(* CODESYS project SPT_Diagnostic.library
   Company: Beckhoff Automation LLC
   DefaultNamespace: SPT_Diagnostic
   Version: 3.3.8
   Placeholder: SPT Diagnostic
   Author: SPT
   Title: SPT Diagnostic

Project tree, tasks and I/O mapping:
  libraries: SPT Base Types, * (Beckhoff Automation LLC); SPT Event Logger, * (Beckhoff Automation LLC); Tc2_EtherCAT, * (Beckhoff Automation GmbH); Tc2_IoFunctions, * (Beckhoff Automation GmbH); Tc2_Standard, * (Beckhoff Automation GmbH); Tc2_System, * (Beckhoff Automation GmbH); Tc2_Utilities, * (Beckhoff Automation GmbH); Tc3_EventLogger, * (Beckhoff Automation GmbH); Tc3_Module, * (Beckhoff Automation GmbH)
  Device Diagnostic/
    DUT/
      data type ST_DeviceInfo
    function block FB_Component_Devices [ST]: Reset, CyclicLogic, CyclicLogic_EtherCat, Update, Initialize, DeviceInfo, LocalAmsNetId
  EtherCat Diagnostic/
    DUT/
      data type ST_EtherCatMaster_Command
      data type ST_EtherCatMaster_Config
      data type ST_EtherCatMaster_HMI
      data type ST_EtherCatMaster_Status
      data type ST_SyncUnitInfo
    function F_EtherCAT_VendorIDtoString [ST]
    function block FB_EtherCatMaster [ST]: CreateEvents, Monitoring, Reset, CyclicLogic, Update, GetSlaveNameByAddr, GetSyncUnitSlaveNames, LookupMasterDevState, LookupSlaveDevState, RaiseAlarmWithStringsAndFlags, RaiseWarningWithStringParameters, SlaveIsPartOfSyncUnit, FB_init, HMICommunication, Initialize, MasterState, SlaveState, EtherCatMasterInfo
    function block FB_EtherCatSyncUnits [ST]: CyclicLogic, SyncUnits, Update, LocalAmsNetId
  Interface/
    interface I_Diagnostic: Update
    interface I_EtherCatSyncUnits: SyncUnits
    interface I_SafetyBase: DependenceFB, OK, SafetyReset
    interface I_SafetyReset: Execute, PulseDuration
    interface I_SafetySimulation: SimulateSafetyDiag, SimulateSafetyState
  Project Information/
    function F_GetCompany [ST]
    function F_GetTitle [ST]
    function F_GetVersion [ST]
  Safety/
    Safety FBs Diagnostic/
      DUT/
        data type E_ComponentSafetyConnection_State
        data type E_ComponentSafetyEdm_State
        data type E_ComponentSafetyEStop_State
        data type E_ComponentSafetyGroup_Diag
        data type E_ComponentSafetyGroup_State
        data type E_ComponentSafetyMon_State
        data type E_ComponentSafetyOrAnd_State
        data type ST_SafetyStateDiag
      Reset Functionblocks/
        function block FB_SafetyResetPulse [ST]: CyclicLogic, Execute, PulseDuration
      function block FB_Component_Safety_AndOrFB [ST]: CyclicLogic, Initialize
      function block FB_Component_Safety_Base [ST]: Reset, CyclicLogic, DependenceFB, OK, SafetyReset, SimulateSafetyDiag, SimulateSafetyState, Initialize
      function block FB_Component_Safety_ConnectionFB [ST]: CreateEvents, Monitoring, Reset, CyclicLogic, Initialize
      function block FB_Component_Safety_EdmFB [ST]: CreateEvents, Monitoring, Reset, CyclicLogic, Initialize
      function block FB_Component_Safety_EstopFB [ST]: CreateEvents, Monitoring, Reset, CyclicLogic, ActiveName, Initialize
      function block FB_Component_Safety_Group [ST]: CreateEvents, Monitoring, Reset, CyclicLogic, AutoResetConnectionFaults, Initialize
      function block FB_Component_Safety_MonFB [ST]: CreateEvents, Monitoring, Reset, CyclicLogic, ActiveAlarm, ActiveName
    Safety Hardware Diagnostic/
  Version/
    global variables Global_Version
  global variables Parameter_Diagnostic
*)

// Device Diagnostic/DUT/ST_DeviceInfo
TYPE ST_DeviceInfo :
	STRUCT
		AmsNetID	   : T_AMSNETID;
		DeviceID	   : UINT;
		DeviceName	   : T_MAXSTRING;
		DeviceType	   : IODEVICETYPES;
		ipDiagnosticFB : I_Diagnostic;
	END_STRUCT
END_TYPE

// EtherCat Diagnostic/DUT/ST_EtherCatMaster_Command
TYPE ST_EtherCatMaster_Command :
	STRUCT
	END_STRUCT
END_TYPE

// EtherCat Diagnostic/DUT/ST_EtherCatMaster_Config
TYPE ST_EtherCatMaster_Config :
	STRUCT
		DeviceInfo : ST_DeviceInfo;
	END_STRUCT
END_TYPE

// EtherCat Diagnostic/DUT/ST_EtherCatMaster_HMI
TYPE ST_EtherCatMaster_HMI :
	STRUCT
		Config	: ST_EtherCatMaster_Config;
		Command : ST_EtherCatMaster_Command;
		Status	: ST_EtherCatMaster_Status;
	END_STRUCT
END_TYPE

// EtherCat Diagnostic/DUT/ST_EtherCatMaster_Status
TYPE ST_EtherCatMaster_Status :
	STRUCT
		EcSlavesState		: ARRAY[0..Parameter_Diagnostic.ETHERCAT_MASTER_SLAVE_MAX] OF ST_EcSlaveState;
		ConfiguredSlaveInfo : ARRAY[0..Parameter_Diagnostic.ETHERCAT_MASTER_SLAVE_MAX] OF ST_EcSlaveConfigData;
		EcSlaveTopologyInfo : ARRAY[0..Parameter_Diagnostic.ETHERCAT_MASTER_SLAVE_MAX] OF ST_TopologyDataEx;
	END_STRUCT
END_TYPE

// EtherCat Diagnostic/DUT/ST_SyncUnitInfo
TYPE ST_SyncUnitInfo :
	STRUCT
		Parent		   : T_MAXSTRING;
		Name		   : STRING(63);
		NumberOfSlaves : UINT;
		Slaves		   : ARRAY[1..Parameter_Diagnostic.ETHERCAT_MASTER_SYNC_UNIT_SLAVE_MAX] OF UINT;
	END_STRUCT
END_TYPE

// Safety/Safety FBs Diagnostic/DUT/E_ComponentSafetyConnection_State
{attribute 'qualified_only'}
{attribute 'strict'}
TYPE E_ComponentSafetyConnection_State : (
		Reset	   := 100,
		Session	   := 101,
		Connection := 102,
		Parameter  := 103,
		Data	   := 104,
		Shutdown   := 105,
		Deactive   := 106
	) USINT;
END_TYPE

// Safety/Safety FBs Diagnostic/DUT/E_ComponentSafetyEdm_State
{attribute 'qualified_only'}
TYPE E_ComponentSafetyEdm_State : (
		Invalid := 0,
		Stop	:= 2,
		Error	:= 4,
		Reset	:= 5,
		MonOff	:= 14,
		MonOn	:= 15
	) USINT;
END_TYPE

// Safety/Safety FBs Diagnostic/DUT/E_ComponentSafetyEStop_State
{attribute 'qualified_only'}
TYPE E_ComponentSafetyEStop_State : (
		Invalid	 := 0,
		Run		 := 1,
		Stop	 := 2,
		Safe	 := 3,
		Error	 := 4,
		Reset	 := 5,
		Start	 := 6,
		DelayOut := 7
	) USINT;
END_TYPE

// Safety/Safety FBs Diagnostic/DUT/E_ComponentSafetyGroup_Diag
{attribute 'qualified_only'}
TYPE E_ComponentSafetyGroup_Diag : (
		NoError		  := 0,
		FbError		  := 1,
		ComError	  := 2,
		ModuleError	  := 3,
		CmpError	  := 4,
		DeactiveError := 5,
		RestartError  := 6
	) UINT;
END_TYPE

// Safety/Safety FBs Diagnostic/DUT/E_ComponentSafetyGroup_State
{attribute 'qualified_only'}
TYPE E_ComponentSafetyGroup_State : (
		Invalid		 := 0,
		Run			 := 1,
		Stop		 := 2,
		Error		 := 4,
		Reset		 := 5,
		Start		 := 6,
		StopError	 := 7,
		Deactive	 := 16,
		WaitComError := 17
	) USINT;
END_TYPE

// Safety/Safety FBs Diagnostic/DUT/E_ComponentSafetyMon_State
{attribute 'qualified_only'}
TYPE E_ComponentSafetyMon_State : (
		Invalid	   := 0,
		Run		   := 1,
		Stop	   := 2,
		Safe	   := 3,
		Error	   := 4,
		Reset	   := 5,
		Start	   := 6,
		ErrorDelay := 7,
		DelayOut   := 8,
		FuncTest   := 9
	) USINT;
END_TYPE

// Safety/Safety FBs Diagnostic/DUT/E_ComponentSafetyOrAnd_State
{attribute 'qualified_only'}
TYPE E_ComponentSafetyOrAnd_State : (
		Invalid := 0,
		Run		:= 1,
		Stop	:= 2,
		Safe	:= 3
	) USINT;
END_TYPE

// Safety/Safety FBs Diagnostic/DUT/ST_SafetyStateDiag
{attribute 'pack_mode' := '1'}
TYPE ST_SafetyStateDiag :
	STRUCT
		State : USINT;
		Diag  : UINT; // **NOT PRESENT ON AND/OR FBs ** For components with USINT as Diag connection, connect first 8 Bit of UINT Diag. Inherited FB is evaluating correct length.
	END_STRUCT
END_TYPE

// Version/Global_Version
{attribute 'TcGenerated'}
{attribute 'no-analysis'}
{attribute 'linkalways'}
// This function has been automatically generated from the project information.
VAR_GLOBAL CONSTANT
	{attribute 'const_non_replaced'}
	stLibVersion_SPT_Diagnostic : ST_LibVersion := (iMajor := 3, iMinor := 3, iBuild := 8, iRevision := 0, nFlags := 1, sVersion := '3.3.8');
END_VAR

// Parameter_Diagnostic
{attribute 'qualified_only'}
VAR_GLOBAL CONSTANT
	UPDATE_TIME : TIME	:= T#500MS; // Start Diagnostic Run every xxx ms, T#0s = deactivated, update needs to manually occur via I_Diagnostic.Upadate()
	DEVICES_MAX : UDINT := 5;		// Max Devices in this System

	// EtherCat
	ETHERCAT_MASTER_START_UP_TIME		: TIME					  := T#1S; // Time to Startup EtherCat Master Diagnostic at initial startup
	ETHERCAT_MASTER_MAX					: UDINT					  := 5;	   // Max EtherCat Masters
	ETHERCAT_MASTER_SLAVE_MAX			: UDINT(1..EC_MAX_SLAVES) := 50;   // Max Slaves per EtherCat Master
	ETHERCAT_MASTER_SYNC_UNIT_MAX		: UDINT					  := 10;   // Max Count of Sync Units per Master
	ETHERCAT_MASTER_SYNC_UNIT_SLAVE_MAX : UDINT					  := 30;   // Max Count of Slaves per Sync Unit

	// Profinet

	// ProfiBus

	// EtherNet

	//...
END_VAR

// Device Diagnostic/FB_Component_Devices
{attribute 'no_explicit_call' := 'do not call this FB directly'}
FUNCTION_BLOCK FB_Component_Devices EXTENDS FB_ComponentBase IMPLEMENTS I_Diagnostic
VAR
	// System Information
	GetLocalAmsNetId : FB_GetLocalAmsNetId;
	GetDeviceIds	 : IOF_GetDeviceIDs;
	DeviceIds		 : ARRAY[0..Parameter_Diagnostic.DEVICES_MAX] OF WORD; //0 = Device counter, 1..X = Device ID's
	GetDeviceType	 : IOF_GetDeviceType;
	GetDeviceName	 : IOF_GetDeviceName;
	GetDeviceNetId	 : IOF_GetDeviceNetId;

	// Instances of Devices
	EtherCatSyncUnits	: FB_EtherCatSyncUnits;																		  // All Sync Units in this runtime
	EtherCatMaster		: ARRAY[1..Parameter_Diagnostic.ETHERCAT_MASTER_MAX] OF FB_EtherCatMaster(EtherCatSyncUnits); //
	EtherCatMasterCount : UDINT(0..Parameter_Diagnostic.ETHERCAT_MASTER_MAX) := 0;									  // Start at 0 to identify existing during Initialzation

	// Properties
	_DeviceInfo	   : ARRAY[1..Parameter_Diagnostic.DEVICES_MAX] OF ST_DeviceInfo;
	_LocalAmsNetId : T_AmsNetId := '';

	// Alarms

	// HMI

	// Sequences
	InitializeSequence : UDINT := 0;
	DeviceNumber	   : UDINT := 1;
	i				   : UDINT := 0; // Iterator
END_VAR

VAR
	// Local
	UpdateOn	: TON;
	UpdateOff	: TON;
	RtrigUpdate : R_TRIG;
END_VAR

//! @summary Clears error flags and error IDs for this component
METHOD PUBLIC Reset : BOOL
Reset := SUPER^.Reset();
IF EtherCatMasterCount >= 1 THEN
	FOR i := 1 TO EtherCatMasterCount DO
		EtherCatMaster[i].Reset();
	END_FOR
END_IF
END_METHOD

//! @summary This method serves as the entry point for all underlying FB logic
METHOD PUBLIC CyclicLogic

//! @description This method should be called cyclically by descendant function blocks by invoking <c>SUPER^.CyclicLogic()</c>.  Alternatively, the contents of this method could be reimplemented entirely in which case a call to this method would not be necessary.
IF NOT _InitComplete THEN
	_InitComplete := Initialize();
	RETURN;
END_IF

// Update Toggle
IF Parameter_Diagnostic.UPDATE_TIME > T#0MS THEN
	UpdateOn(IN := NOT UpdateOff.Q, PT := Parameter_Diagnostic.UPDATE_TIME);
	UpdateOff(IN := UpdateOn.Q, PT := Parameter_Diagnostic.UPDATE_TIME);
	RtrigUpdate(CLK := UpdateOn.Q);
END_IF

// Cyclic Logics
CyclicLogic_EtherCat();
SUPER^.CyclicLogic();

// Error Status Update of all Devices
_Error := FALSE;
_Busy  := FALSE;
IF EtherCatMasterCount >= 1 THEN
	FOR i := 1 TO EtherCatMasterCount DO
		IF _CurrentAlarmSeverity < EtherCatMaster[i].CurrentAlarmSeverity THEN
			_CurrentAlarmSeverity := EtherCatMaster[i].CurrentAlarmSeverity;
		END_IF

		_Error := _Error OR EtherCatMaster[i].Error;
		_Busy  := _Busy OR EtherCatMaster[i].Busy;
		IF EtherCatMaster[i].ErrorID <> 0 AND _ErrorID = 0 THEN
			_ErrorID := EtherCatMaster[i].ErrorID;
		END_IF
	END_FOR
END_IF
END_METHOD

METHOD CyclicLogic_EtherCat
// Get all Sync Units in Runtime
EtherCatSyncUnits.LocalAmsNetId := _LocalAmsNetId;
EtherCatSyncUnits.CyclicLogic();

// Call Cyclic
IF EtherCatMasterCount >= 1 THEN
	FOR i := 1 TO EtherCatMasterCount DO
		// Update
		IF RtrigUpdate.Q THEN
			EtherCatMaster[i].Update();
		END_IF

		// Cyclic Call
		EtherCatMaster[i].CyclicLogic();
	END_FOR
END_IF
END_METHOD

METHOD Update
IF EtherCatMasterCount >= 1 THEN
	FOR i := 1 TO EtherCatMasterCount DO
		EtherCatMaster[i].Update();
	END_FOR
END_IF
END_METHOD

//! @summary Basic component initialization logic
METHOD PROTECTED Initialize : BOOL;
//! @description This method is called by <c>CyclicLogic()</c> as required
VAR_INST
	AllDevicesInitialized : BOOL := FALSE;
END_VAR
Initialize := FALSE;
IF _Simulate THEN
	Initialize := SUPER^.Initialize();
	RETURN;
END_IF

// Call FBs
GetLocalAmsNetId(tTimeOut := T#1S);
GetDeviceIds(NETID := _LocalAmsNetId, TMOUT := T#1S);
GetDeviceName(NETID := _LocalAmsNetId, TMOUT := T#1S);
GetDeviceNetId(NETID := _LocalAmsNetId, TMOUT := T#1S);
GetDeviceType(NETID := _LocalAmsNetId, TMOUT := T#1S);

// Init Sequence
CASE InitializeSequence OF
	0: // Get local AmsNet-Id
		GetLocalAmsNetId.bExecute := TRUE;
		IF GetLocalAmsNetId.bBusy THEN
			InitializeSequence := InitializeSequence + 10;
		END_IF

	10: // Get local AmsNet-Id
		IF NOT GetLocalAmsNetId.bBusy AND NOT GetLocalAmsNetId.bError THEN
			_LocalAmsNetId	   := GetLocalAmsNetId.AddrString;
			InitializeSequence := InitializeSequence + 10;
		END_IF

		IF GetLocalAmsNetId.bError THEN
			_ErrorID := GetLocalAmsNetId.nErrId;
			Trace('Init Failed - GetLocalAmsNetId!');
			InitializeSequence := 999;
		END_IF

	20: // Get all Devices in this System
		GetDeviceIds.LEN	  := SIZEOF(DeviceIds);
		GetDeviceIds.DESTADDR := ADR(DeviceIds);
		GetDeviceIds.START	  := TRUE;
		IF GetDeviceIds.BUSY THEN
			GetDeviceIds.START := FALSE;
			InitializeSequence := InitializeSequence + 10;
		END_IF

	30: // Get all Devices in this System
		IF NOT GetDeviceIds.BUSY AND NOT GetDeviceIds.ERR THEN
			// Devices found
			IF (DeviceIDs[0] > 0) AND NOT _Simulate THEN
				// Map device Ids
				FOR i := 1 TO DeviceIDs[0] DO
					IF i <= Parameter_Diagnostic.DEVICES_MAX THEN
						_DeviceInfo[i].DeviceID := DeviceIDs[i];
					ELSE
						Trace('Init Failed - find IO Devices, Diagnostic, not enough Devices foreseen! Increase DEVICES_MAX');
						InitializeSequence := 999;
						EXIT;
					END_IF
				END_FOR

				InitializeSequence := InitializeSequence + 10;
			ELSE
				_Simulate		   := TRUE; // No devices found = activate simulation mode
				InitializeSequence := 1000;
			END_IF
		END_IF

		IF GetDeviceIds.ERR THEN
			_ErrorID := GetDeviceIds.ERRID;
			Trace('Init Failed - GetDeviceIds!');
			InitializeSequence := 999;
		END_IF

	40: // Get Device Names
		GetDeviceName.DEVICEID := DeviceIDs[DeviceNumber];
		GetDeviceName.START	   := TRUE;
		IF GetDeviceName.BUSY THEN
			GetDeviceName.START := FALSE;
			InitializeSequence	:= InitializeSequence + 10;
		END_IF

	50: // Get Device Names
		IF NOT GetDeviceName.BUSY AND NOT GetDeviceName.ERR THEN
			// Next Device
			_DeviceInfo[DeviceNumber].DeviceName := GetDeviceName.DEVICENAME;
			DeviceNumber						 := DeviceNumber + 1;
			IF (DeviceIDs[DeviceNumber] <> 0) THEN
				InitializeSequence := InitializeSequence - 10;
			ELSE
				DeviceNumber	   := 1;
				InitializeSequence := InitializeSequence + 10;
			END_IF
		END_IF

		IF GetDeviceName.ERR THEN
			_ErrorID := GetDeviceName.ERRID;
			Trace('Init Failed - GetDeviceName!');
			InitializeSequence := 999;
		END_IF

	60: // Get Device NetIds
		GetDeviceNetId.DEVICEID := DeviceIDs[DeviceNumber];
		GetDeviceNetId.START	:= TRUE;
		IF GetDeviceNetId.BUSY THEN
			GetDeviceNetId.START := FALSE;
			InitializeSequence	 := InitializeSequence + 10;
		END_IF

	70: // Get Device NetIds
		IF NOT GetDeviceNetId.BUSY AND NOT GetDeviceNetId.ERR THEN
			// Next Device
			_DeviceInfo[DeviceNumber].AmsNetID := GetDeviceNetId.DeviceNetId;
			DeviceNumber					   := DeviceNumber + 1;
			IF (DeviceIDs[DeviceNumber] <> 0) THEN
				InitializeSequence := InitializeSequence - 10;
			ELSE
				DeviceNumber	   := 1;
				InitializeSequence := InitializeSequence + 10;
			END_IF
		END_IF

		IF GetDeviceNetId.ERR THEN
			_ErrorID := GetDeviceNetId.ERRID;
			Trace('Init Failed - GetDeviceNetId!');
			InitializeSequence := 999;
		END_IF

	80: // Get Device Types
		GetDeviceType.DEVICEID := DeviceIDs[DeviceNumber];
		GetDeviceType.START	   := TRUE;
		IF GetDeviceType.BUSY THEN
			GetDeviceType.START := FALSE;
			InitializeSequence	:= InitializeSequence + 10;
		END_IF

	90: // Get Device Types
		IF NOT GetDeviceType.BUSY AND NOT GetDeviceType.ERR THEN
			// Next Device
			_DeviceInfo[DeviceNumber].DeviceType := GetDeviceType.IODeviceType;
			DeviceNumber						 := DeviceNumber + 1;
			IF (DeviceIDs[DeviceNumber] <> 0) THEN
				InitializeSequence := InitializeSequence - 10;
			ELSE
				DeviceNumber	   := 1;
				InitializeSequence := InitializeSequence + 10;
			END_IF
		END_IF

		IF GetDeviceType.ERR THEN
			_ErrorID := GetDeviceType.ERRID;
			Trace('Init Failed - GetDeviceType!');
			InitializeSequence := 999;
		END_IF

	100: // Initalize all Devices found
		FOR i := 1 TO DeviceIDs[0] DO
			CASE DeviceInfo[i].DeviceType OF
				IODEVICETYPES.IODEVICETYPE_ETHERCAT:
					EtherCatMasterCount := EtherCatMasterCount + 1;
					IF EtherCatMasterCount <= Parameter_Diagnostic.ETHERCAT_MASTER_MAX THEN
						EtherCatMaster[EtherCatMasterCount].EtherCatMasterInfo REF= _DeviceInfo[i];
						EtherCatMaster[EtherCatMasterCount].Name			   := DeviceInfo[i].DeviceName;
						DeviceInfo[i].ipDiagnosticFB						   := EtherCatMaster[EtherCatMasterCount];
					ELSE
						Trace('Init Failed - not enough EtherCat Master Diagnostics Instances! Increase ETHERCAT_MASTER_MAX');
						InitializeSequence := 999;
					END_IF

			ELSE
				Trace(CONCAT('Warning - Device Diagnostics for this Device does not exist! ', DeviceInfo[i].DeviceName));
			END_CASE
		END_FOR

		// No error during initialization
		IF InitializeSequence <> 999 THEN
			InitializeSequence := InitializeSequence + 10;
		END_IF

	110: // Initalize all Devices found
		AllDevicesInitialized := TRUE;

		// Init all EtherCat Master Devices
		IF EtherCatMasterCount >= 1 THEN
			FOR i := 1 TO EtherCatMasterCount DO
				EtherCatMaster[i].CyclicLogic();
				AllDevicesInitialized := AllDevicesInitialized AND EtherCatMaster[i].InitComplete;
			END_FOR
		END_IF

		IF AllDevicesInitialized THEN
			InitializeSequence := 1000;
		END_IF

	1000: // Initialize the Base
		IF SUPER^.Initialize() THEN
			Initialize := TRUE;
			_Error	   := FALSE;
			_Busy	   := FALSE;
		END_IF

	999:
		_Error := TRUE;
		_Busy  := FALSE;
END_CASE
END_METHOD

{analysis -29}
PROPERTY DeviceInfo : REFERENCE TO ARRAY[1..Parameter_Diagnostic.DEVICES_MAX] OF ST_DeviceInfo
GET
DeviceInfo REF= _DeviceInfo;
END_GET
END_PROPERTY

PROPERTY LocalAmsNetId : T_AmsNetId
GET
LocalAmsNetId := _LocalAmsNetId;
END_GET
END_PROPERTY

END_FUNCTION_BLOCK

// Interface/I_Diagnostic
INTERFACE I_Diagnostic EXTENDS I_BaseFB

METHOD Update
VAR_INPUT
END_VAR
END_METHOD

END_INTERFACE

// EtherCat Diagnostic/FB_EtherCatSyncUnits
{attribute 'no_explicit_call' := 'do not call this FB directly'}
FUNCTION_BLOCK FB_EtherCatSyncUnits EXTENDS FB_CyclicFB IMPLEMENTS I_EtherCatSyncUnits
VAR
	(* Sequence *)
	SyncUnitSequence : UINT;

	(* Local *)
	GetSyncUnitOids			  : ADSRDWRT;
	GetAllSyncUnitSlaveAddr	  : FB_EcGetAllSyncUnitSlaveAddr;
	ipSyncUnitComObject		  : ITComObject;
	ipSyncUnitParentComObject : ITComObject;
	SyncUnitCount			  : DWORD;
	i						  : DWORD; // Iterator
	SyncUnitParentOid		  : OTCID;
	SyncUnitOids			  : ARRAY[1..Parameter_Diagnostic.ETHERCAT_MASTER_SYNC_UNIT_MAX] OF OTCID;

	(* Properties *)
	_SyncUnits	   : ARRAY[1..Parameter_Diagnostic.ETHERCAT_MASTER_SYNC_UNIT_MAX] OF ST_SyncUnitInfo;
	_LocalAmsNetId : T_AmsNetId;
END_VAR

VAR CONSTANT
	SYNC_UNIT_CLASS_ID : CLSID := STRING_TO_GUID('03020004-0000-0000-F000-000000000064');
END_VAR

METHOD PUBLIC CyclicLogic
VAR_INST
	tempName		 : STRING(63);
	SyncUnitIterator : UINT := 1;
END_VAR
{analysis -19}
{analysis -07}

// Call FBs
GetSyncUnitOids(NETID := _LocalAmsNetId);
GetAllSyncUnitSlaveAddr(sNetId := _LocalAmsNetId);

// Sequence
CASE SyncUnitSequence OF
	0: // Wait for start
		GetSyncUnitOids.WRTRD			 := FALSE;
		GetAllSyncUnitSlaveAddr.bExecute := FALSE;
		SyncUnitIterator				 := 1;

	10: // Get Sync Unit Count

		// Reset for restart
		_Error	 := FALSE;
		_ErrorID := 0;

		// Get Sync Unit Count
		GetSyncUnitOids.PORT	 := 10;
		GetSyncUnitOids.IDXGRP	 := 16#201;
		GetSyncUnitOids.IDXOFFS	 := 16#01;
		GetSyncUnitOids.WRITELEN := SIZEOF(SYNC_UNIT_CLASS_ID);
		GetSyncUnitOids.SRCADDR	 := ADR(SYNC_UNIT_CLASS_ID);
		GetSyncUnitOids.READLEN	 := SIZEOF(SyncUnitCount);
		GetSyncUnitOids.DESTADDR := ADR(SyncUnitCount);
		GetSyncUnitOids.WRTRD	 := TRUE;
		IF GetSyncUnitOids.BUSY THEN
			SyncUnitSequence := SyncUnitSequence + 10;
		END_IF

	20: // Get Sync Unit Count
		IF NOT GetSyncUnitOids.BUSY AND NOT GetSyncUnitOids.ERR THEN
			// Byte Adjustment
			SyncUnitCount		  := SyncUnitCount / 4;
			GetSyncUnitOids.WRTRD := FALSE;
			IF SyncUnitCount <= Parameter_Diagnostic.ETHERCAT_MASTER_SYNC_UNIT_MAX THEN // Check configuration and space
				IF SyncUnitCount > 0 THEN												// Only if Sync Unit exist - run diag
					SyncUnitSequence := SyncUnitSequence + 10;
				ELSE
					SyncUnitSequence := 0;
				END_IF
			ELSE
				SyncUnitSequence := 999;
				_ErrorID		 := SyncUnitCount;
				Trace('FB_EtherCatSyncUnits - not enough Sync Units foreseen! Increase ETHERCAT_MASTER_SYNC_UNIT_MAX');
			END_IF
		END_IF

		IF GetSyncUnitOids.ERR THEN
			_ErrorID		 := GetSyncUnitOids.ERRID;
			SyncUnitSequence := 999;
		END_IF

	30: // Get Sync Unit Oids
		GetSyncUnitOids.PORT	 := 10;
		GetSyncUnitOids.IDXGRP	 := 16#201;
		GetSyncUnitOids.IDXOFFS	 := 16#02;
		GetSyncUnitOids.WRITELEN := SIZEOF(SYNC_UNIT_CLASS_ID);
		GetSyncUnitOids.SRCADDR	 := ADR(SYNC_UNIT_CLASS_ID);
		GetSyncUnitOids.READLEN	 := (SIZEOF(OTCID) * SyncUnitCount);
		GetSyncUnitOids.DESTADDR := ADR(SyncUnitOids);
		GetSyncUnitOids.WRTRD	 := TRUE;
		IF GetSyncUnitOids.BUSY THEN
			SyncUnitSequence := SyncUnitSequence + 10;
		END_IF

	40: // Get Sync Unit Oids
		IF NOT GetSyncUnitOids.BUSY AND NOT GetSyncUnitOids.ERR THEN
			GetSyncUnitOids.WRTRD := FALSE;
			SyncUnitSequence	  := SyncUnitSequence + 10;
		END_IF

		IF GetSyncUnitOids.ERR THEN
			_ErrorID		 := GetSyncUnitOids.ERRID;
			SyncUnitSequence := 999;
		END_IF

	50: // Get EtherCat Master and Name of Sync Unit
		FOR i := 1 TO SyncUnitCount DO
			// Get Sync Unit
			FW_ObjMgr_GetObjectInstance(SyncUnitOids[i], TC_GLOBAL_IID_LIST.IID_ITComObject, ADR(ipSyncUnitComObject));
			IF ipSyncUnitComObject <> 0 THEN
				ipSyncUnitComObject.TcGetObjectName(objName := ADR(_SyncUnits[i].Name), nameLen := SIZEOF(_SyncUnits[i].Name));
				F_EcGetSyncUnitName(SyncUnitOids[i], sSyncUnitName => tempName);
				tempName		   := CONCAT(tempName, ' - ');
				_SyncUnits[i].Name := CONCAT(tempName, _SyncUnits[i].Name);

				// Get Parent
				ipSyncUnitComObject.TcGetParentObjId(SyncUnitParentOid);
				FW_ObjMgr_GetObjectInstance(SyncUnitParentOid, TC_GLOBAL_IID_LIST.IID_ITComObject, ADR(ipSyncUnitParentComObject));
				IF ipSyncUnitParentComObject <> 0 THEN
					ipSyncUnitParentComObject.TcGetObjectName(objName := ADR(_SyncUnits[i].Parent), nameLen := SIZEOF(_SyncUnits[i].Parent));
					FW_SafeRelease(pipUnk := ADR(ipSyncUnitParentComObject));
				END_IF

				FW_SafeRelease(pipUnk := ADR(ipSyncUnitComObject));
			END_IF
		END_FOR

		SyncUnitSequence := SyncUnitSequence + 10;

	60: // Get all sync Unit Slaves 
		IF SyncUnitIterator > Parameter_Diagnostic.ETHERCAT_MASTER_SYNC_UNIT_MAX THEN
			SyncUnitSequence := 0; // All Sync units searched
		ELSE
			IF SyncUnitOids[SyncUnitIterator] = 0 THEN
				SyncUnitSequence := 0; // Done
			ELSE
				GetAllSyncUnitSlaveAddr.nObjectId := SyncUnitOids[SyncUnitIterator];
				GetAllSyncUnitSlaveAddr.pAddrBuf  := ADR(_SyncUnits[SyncUnitIterator].Slaves);
				GetAllSyncUnitSlaveAddr.cbBufLen  := SIZEOF(_SyncUnits[SyncUnitIterator].Slaves);
				GetAllSyncUnitSlaveAddr.bExecute  := TRUE;
				IF GetAllSyncUnitSlaveAddr.bBusy THEN
					GetAllSyncUnitSlaveAddr.bExecute := FALSE;
					SyncUnitSequence				 := SyncUnitSequence + 10;
				END_IF
			END_IF
		END_IF

	70: // Get all sync Unit Slaves
		IF NOT GetAllSyncUnitSlaveAddr.bBusy AND NOT GetAllSyncUnitSlaveAddr.bError THEN
			_SyncUnits[SyncUnitIterator].NumberOfSlaves := GetAllSyncUnitSlaveAddr.nSlaves;
			SyncUnitIterator							:= SyncUnitIterator + 1;
			IF _SyncUnits[SyncUnitIterator].NumberOfSlaves <= Parameter_Diagnostic.ETHERCAT_MASTER_SYNC_UNIT_SLAVE_MAX THEN
				SyncUnitSequence := SyncUnitSequence - 10;
			ELSE
				SyncUnitSequence := 999;
				_ErrorID		 := _SyncUnits[SyncUnitIterator].NumberOfSlaves;
				Trace('FB_EtherCatSyncUnits - not enough slaves per Sync Units foreseen! Increase ETHERCAT_MASTER_SYNC_UNIT_SLAVE_MAX');
			END_IF
		END_IF

		IF GetAllSyncUnitSlaveAddr.bError THEN
			_ErrorID		 := GetAllSyncUnitSlaveAddr.nErrId;
			SyncUnitSequence := 999;
		END_IF

	999: // Error
		SyncUnitSequence := 0;
		_Error			 := TRUE;
		Trace('FB_EtherCatSyncUnits - Error get Sync Units Sequence!');
END_CASE

_Busy := SyncUnitSequence <> 0;
END_METHOD

PROPERTY SyncUnits : REFERENCE TO ARRAY[1..Parameter_Diagnostic.ETHERCAT_MASTER_SYNC_UNIT_MAX] OF ST_SyncUnitInfo
GET
SyncUnits REF= _SyncUnits;
END_GET
END_PROPERTY

METHOD Update
IF NOT _Busy THEN
	SyncUnitSequence := 10;
END_IF
END_METHOD

PROPERTY LocalAmsNetId : T_AmsNetId
SET
_LocalAmsNetId := LocalAmsNetId;
END_SET
END_PROPERTY

END_FUNCTION_BLOCK

// Interface/I_EtherCatSyncUnits
INTERFACE I_EtherCatSyncUnits EXTENDS I_Diagnostic

PROPERTY SyncUnits : REFERENCE TO ARRAY[1..Parameter_Diagnostic.ETHERCAT_MASTER_SYNC_UNIT_MAX] OF ST_SyncUnitInfo
GET
END_GET
END_PROPERTY

END_INTERFACE

// EtherCat Diagnostic/FB_EtherCatMaster
{attribute 'no_explicit_call' := 'do not call this FB directly'}
FUNCTION_BLOCK FB_EtherCatMaster EXTENDS FB_ComponentBase IMPLEMENTS I_Diagnostic
VAR
	(* Internal Variables *)
	EcGetMasterDevState	 : FB_EcGetMasterDevState;
	GetSlaveTopologyInfo : FB_EcGetSlaveTopologyInfo;
	EcGetAllSlaveStates	 : FB_EcGetAllSlaveStates;
	GetConfiguredSlaves	 : FB_EcGetConfSlaves;
	EcSlavesState		 : ARRAY[0..Parameter_Diagnostic.ETHERCAT_MASTER_SLAVE_MAX] OF ST_EcSlaveState;
	ConfiguredSlaveInfo	 : ARRAY[0..Parameter_Diagnostic.ETHERCAT_MASTER_SLAVE_MAX] OF ST_EcSlaveConfigData;
	EcSlaveTopologyInfo	 : ARRAY[0..Parameter_Diagnostic.ETHERCAT_MASTER_SLAVE_MAX] OF ST_TopologyDataEx;
	SyncUnits			 : REFERENCE TO ARRAY[1..Parameter_Diagnostic.ETHERCAT_MASTER_SYNC_UNIT_MAX] OF ST_SyncUnitInfo;
	MasterDevState		 : WORD;
	SlaveCount			 : UINT;
	CfgSlaveCount		 : UINT;

	(* Properties *)
	_EtherCatMasterInfo : REFERENCE TO ST_DeviceInfo;

	(* HMI *)
	EtherCatMaster_HMI : ST_EtherCatMaster_HMI;

	(* Sync Units *)
	ipEtherCatSyncUnits : I_EtherCatSyncUnits;

	(* Sequence *)
	SlaveSeq	: UINT;
	MasterSeq	: UINT;
	SyncUnitSeq : UINT;

	(* Alarms *)
	MasterAlarms	 : ARRAY[1..MASTER_ALARM_COUNT] OF FB_TcAlarm;
	SlaveErrors		 : ARRAY[0..Parameter_Diagnostic.ETHERCAT_MASTER_SLAVE_MAX] OF FB_TcAlarm;
	SlaveWarnings	 : ARRAY[0..Parameter_Diagnostic.ETHERCAT_MASTER_SLAVE_MAX] OF FB_TcAlarm;
	SyncUnitWarnings : ARRAY[1..Parameter_Diagnostic.ETHERCAT_MASTER_SYNC_UNIT_MAX] OF FB_TcAlarm;
END_VAR

VAR CONSTANT
	MASTER_ALARM_COUNT : UDINT := 3;
	STRING_LEN		   : INT   := 80;
END_VAR

METHOD PROTECTED CreateEvents
//! @description This method is called by <c>Initialize()</c> as required
VAR_INST
	tempName   : STRING;
	SourceInfo : FB_TcSourceInfo;
	i		   : UDINT;
END_VAR
F_CreateAllEventsInClass(Alarms		:= MasterAlarms,
						 ClassSize	:= SIZEOF(TC_EVENTS.EtherCatMaster),
						 pInitEvent := ADR(TC_EVENTS.EtherCatMaster.InitReferenceEvent),
						 Prefix		:= Name);

SUPER^.CreateEvents();

// Create SyncUnit and Slave Alarms
FOR i := 0 TO Parameter_Diagnostic.ETHERCAT_MASTER_SLAVE_MAX DO
	SourceInfo.sName := CONCAT(CONCAT(THIS^.Name, ' - '), ConfiguredSlaveInfo[i].sName);
	SlaveErrors[i].CreateEx(stEventEntry := TC_EVENTS.EtherCatSlave.SlaveError, 0, SourceInfo);
	SlaveWarnings[i].CreateEx(stEventEntry := TC_EVENTS.EtherCatSlave.SlaveWarning, 0, SourceInfo);
END_FOR

FOR i := 1 TO Parameter_Diagnostic.ETHERCAT_MASTER_SYNC_UNIT_MAX DO
	SourceInfo.sName := CONCAT(CONCAT(THIS^.Name, ' - '), ConfiguredSlaveInfo[i].sName);
	SyncUnitWarnings[i].CreateEx(stEventEntry := TC_EVENTS.SyncUnit.SyncUnitWarning, 0, SourceInfo);
END_FOR
END_METHOD

//! Provides basic error detection and event handling for this component
METHOD PROTECTED Monitoring
(*! @descriptionThis method is called cyclically by <c>CyclicLogic()</c>*)
VAR_INST
	Error1 : BOOL;
	Error2 : BOOL;
	Error3 : BOOL;
END_VAR
SUPER^.Monitoring();

(* EtherCat Master Messages *)

// Raised in Master Sequence

(* EtherCat Slave Messages *)

// Raised in Slave Sequence

(* Alarm Severity of EtherCat Master Device *)
_CurrentAlarmSeverity := F_GetMaxSeverityRaised(Alarms := MasterAlarms, CurrentSeverity := _CurrentAlarmSeverity);
_CurrentAlarmSeverity := F_GetMaxSeverityRaised(Alarms := SlaveErrors, CurrentSeverity := _CurrentAlarmSeverity);
_CurrentAlarmSeverity := F_GetMaxSeverityRaised(Alarms := SlaveWarnings, CurrentSeverity := _CurrentAlarmSeverity);
_CurrentAlarmSeverity := F_GetMaxSeverityRaised(Alarms := SyncUnitWarnings, CurrentSeverity := _CurrentAlarmSeverity);
END_METHOD

//! @summary Clears error flags and error IDs for this component
METHOD PUBLIC Reset : BOOL
F_ClearAllEventsInClass(MasterAlarms);
F_ClearAllEventsInClass(SlaveErrors);
F_ClearAllEventsInClass(SlaveWarnings);
F_ClearAllEventsInClass(SyncUnitWarnings);
SlaveSeq  := 0;
MasterSeq := 0;
_Error	  := FALSE;
_ErrorID  := 0;
_Busy	  := FALSE;
Reset	  := SUPER^.Reset();
END_METHOD

//! @summary This method serves as the entry point for all underlying FB logic
METHOD PUBLIC CyclicLogic

//! @description This method should be called cyclically by descendant function blocks by invoking <c>SUPER^.CyclicLogic()</c>.  Alternatively, the contents of this method could be reimplemented entirely in which case a call to this method would not be necessary.
IF NOT _InitComplete THEN
	_InitComplete := Initialize();
	RETURN;
END_IF

(* Main Component Signals *)
IF _Simulate THEN
	_Busy	 := FALSE;
	_Error	 := FALSE;
	_ErrorID := 0;
ELSE
	// Master State
	MasterState();

	// Slave State
	SlaveState();

	// Super
	_Busy := SlaveSeq <> 0 OR MasterSeq <> 0; // Sequence running
	SUPER^.CyclicLogic();
END_IF
END_METHOD

METHOD Update
IF NOT _Busy THEN
	// Start Master and Slave Diagnostics Sequence
	MasterSeq := 10;
	SlaveSeq  := 10;
END_IF
END_METHOD

METHOD PRIVATE GetSlaveNameByAddr : STRING(31)
VAR_INPUT
	Addr : UINT;
END_VAR

VAR_INST
	Slave : UDINT;
END_VAR
GetSlaveNameByAddr := '';
FOR Slave := 0 TO Parameter_Diagnostic.ETHERCAT_MASTER_SLAVE_MAX DO
	IF ConfiguredSlaveInfo[Slave].nAddr = Addr THEN
		GetSlaveNameByAddr := ConfiguredSlaveInfo[Slave].sName;
		RETURN;
	END_IF
END_FOR
END_METHOD

METHOD PRIVATE GetSyncUnitSlaveNames
VAR_INPUT
	SyncUnit : ST_SyncUnitInfo;
END_VAR

VAR_INST
	i						  : UDINT;
	j						  : UDINT;
	TempSlavesInSyncUnitPartA : STRING;
	TempSlavesInSyncUnitPartB : STRING;
	TempSlaveMessage		  : STRING;
END_VAR

VAR_OUTPUT
	SlavesInSyncUnitPartA : STRING;
	SlavesInSyncUnitPartB : STRING;
END_VAR
TempSlavesInSyncUnitPartA := '';
TempSlavesInSyncUnitPartB := '';
FOR i := 1 TO Parameter_Diagnostic.ETHERCAT_MASTER_SYNC_UNIT_SLAVE_MAX DO
	FOR j := 1 TO Parameter_Diagnostic.ETHERCAT_MASTER_SLAVE_MAX DO
		IF SyncUnit.Slaves[i] <> 0 THEN
			IF SyncUnit.Slaves[i] = ConfiguredSlaveInfo[j].nAddr THEN
				IF LEN(ConfiguredSlaveInfo[j].sName) > 0 THEN
					TempSlaveMessage := CONCAT(ConfiguredSlaveInfo[j].sName, ', ');
					IF (LEN(TempSlaveMessage) + LEN(TempSlavesInSyncUnitPartA)) <= STRING_LEN THEN
						TempSlavesInSyncUnitPartA := CONCAT(TempSlavesInSyncUnitPartA, TempSlaveMessage);
					ELSIF (LEN(TempSlaveMessage) + LEN(TempSlavesInSyncUnitPartB)) <= STRING_LEN THEN
						TempSlavesInSyncUnitPartB := CONCAT(TempSlavesInSyncUnitPartB, TempSlaveMessage);
					END_IF
				END_IF
			END_IF
		END_IF
	END_FOR
END_FOR

SlavesInSyncUnitPartA := TempSlavesInSyncUnitPartA;
SlavesInSyncUnitPartB := TempSlavesInSyncUnitPartB;
END_METHOD

METHOD PROTECTED LookupMasterDevState : STRING
VAR_INPUT
	State : UINT;
END_VAR

VAR_OUTPUT
	TypeError	: BOOL;
	TypeWarning : BOOL;
END_VAR
TypeError	:= FALSE;
TypeWarning := FALSE;
IF State.0 THEN
	TypeError			 := TRUE;
	LookupMasterDevState := 'Link error';
ELSIF State.1 THEN
	TypeError			 := TRUE;
	LookupMasterDevState := 'I/O locked after link error (I/O reset required)';
ELSIF State.2 THEN
	TypeError			 := TRUE;
	LookupMasterDevState := 'Link error (redundancy adapter)';
ELSIF State.3 THEN
	TypeError			 := TRUE;
	LookupMasterDevState := 'Missing one frame (redundancy mode)';
ELSIF State.4 THEN
	TypeError			 := TRUE;
	LookupMasterDevState := 'Out of send resources (I/O reset required)';
ELSIF State.5 THEN
	TypeError			 := TRUE;
	LookupMasterDevState := 'Watchdog triggered';
ELSIF State.6 THEN
	TypeError			 := TRUE;
	LookupMasterDevState := 'Ethernet driver (miniport) NOT found';
ELSIF State.7 THEN
	TypeWarning			 := TRUE;
	LookupMasterDevState := 'I/O reset active';
ELSIF State.8 THEN
	TypeWarning			 := TRUE;
	LookupMasterDevState := 'At least one device in INIT state';
ELSIF State.9 THEN
	TypeWarning			 := TRUE;
	LookupMasterDevState := 'At least one device in PRE-OP state';
ELSIF State.10 THEN
	TypeWarning			 := TRUE;
	LookupMasterDevState := 'At least one device in SAFE-OP state';
ELSIF State.11 THEN
	TypeWarning			 := TRUE;
	LookupMasterDevState := 'At least one device indicates an error state';
ELSIF State.12 THEN
	TypeError			 := TRUE;
	LookupMasterDevState := 'DC not in sync';
ELSE
	TypeWarning			 := TRUE;
	LookupMasterDevState := 'State not found';
END_IF
END_METHOD

METHOD PROTECTED LookupSlaveDevState : STRING
VAR_INPUT
	Slave : UDINT;
END_VAR

VAR_INST
	DiagByte				: BYTE;
	BitMaskDiag				: BYTE := 16#0F;
	tempLookupSlaveDevState : STRING;
END_VAR
//_____________________________________________________________________________________________________

(* State *)
BitMaskDiag := 16#0F;
DiagByte	:= EcSlavesState[Slave].deviceState AND BitMaskDiag;
CASE DiagByte OF
	EC_DEVICE_STATE_INIT:
		tempLookupSlaveDevState := 'Init';

	EC_DEVICE_STATE_PREOP:
		tempLookupSlaveDevState := 'Pre-op';

	EC_DEVICE_STATE_BOOTSTRAP:
		tempLookupSlaveDevState := 'Boot';

	EC_DEVICE_STATE_SAFEOP:
		tempLookupSlaveDevState := 'Safe-op';

	EC_DEVICE_STATE_OP:
		tempLookupSlaveDevState := 'OP';

ELSE
	tempLookupSlaveDevState := '';
END_CASE

(* Additional State Bits *)
IF EcSlavesState[Slave].deviceState.4 THEN //EC_DEVICE_STATE_ERROR
	tempLookupSlaveDevState := CONCAT(tempLookupSlaveDevState, ' - ');
	tempLookupSlaveDevState := CONCAT(tempLookupSlaveDevState, 'State machine error in the EtherCAT slave');
END_IF

IF EcSlavesState[Slave].deviceState.5 THEN //EC_DEVICE_STATE_INVALID_VPRS
	tempLookupSlaveDevState := CONCAT(tempLookupSlaveDevState, ' - ');
	tempLookupSlaveDevState := CONCAT(tempLookupSlaveDevState, 'Invalid vendor ID');
END_IF

IF EcSlavesState[Slave].deviceState.6 THEN //EC_DEVICE_STATE_INITCMD_ERROR
	tempLookupSlaveDevState := CONCAT(tempLookupSlaveDevState, ' - ');
	tempLookupSlaveDevState := CONCAT(tempLookupSlaveDevState, 'Error during sending of initialization commands');
END_IF

IF EcSlavesState[Slave].deviceState.7 THEN //EC_DEVICE_STATE_DISABLED
	tempLookupSlaveDevState := CONCAT(tempLookupSlaveDevState, ' - ');
	tempLookupSlaveDevState := CONCAT(tempLookupSlaveDevState, 'Slave is disabled');
END_IF

//_____________________________________________________________________________________________________

(* Link States *)
IF EcSlavesState[Slave].linkState.0 THEN //EC_LINK_STATE_NOT_PRESENT
	tempLookupSlaveDevState := CONCAT(tempLookupSlaveDevState, ' - ');
	tempLookupSlaveDevState := CONCAT(tempLookupSlaveDevState, 'No EtherCAT communication with the EtherCAT slave');
END_IF

IF EcSlavesState[Slave].linkState.1 THEN //EC_LINK_STATE_LINK_WITHOUT_COMM
	tempLookupSlaveDevState := CONCAT(tempLookupSlaveDevState, ' - ');
	tempLookupSlaveDevState := CONCAT(tempLookupSlaveDevState, 'Error AT port X');
END_IF

IF EcSlavesState[Slave].linkState.2 THEN //EC_LINK_STATE_MISSING_LINK
	tempLookupSlaveDevState := CONCAT(tempLookupSlaveDevState, ' - ');
	tempLookupSlaveDevState := CONCAT(tempLookupSlaveDevState, 'Missing link AT port X');
END_IF

IF EcSlavesState[Slave].linkState.3 THEN //EC_LINK_STATE_ADDITIONAL_LINK
	tempLookupSlaveDevState := CONCAT(tempLookupSlaveDevState, ' - ');
	tempLookupSlaveDevState := CONCAT(tempLookupSlaveDevState, 'Additional link AT port X');
END_IF

(* Additional State Bits *)
IF EcSlavesState[Slave].linkState.4 THEN //EC_LINK_STATE_PORT_A
	tempLookupSlaveDevState := CONCAT(tempLookupSlaveDevState, ' - ');
	tempLookupSlaveDevState := CONCAT(tempLookupSlaveDevState, 'Port 0');
END_IF

IF EcSlavesState[Slave].linkState.5 THEN //EC_LINK_STATE_PORT_B
	tempLookupSlaveDevState := CONCAT(tempLookupSlaveDevState, ' - ');
	tempLookupSlaveDevState := CONCAT(tempLookupSlaveDevState, 'Port 1');
END_IF

IF EcSlavesState[Slave].linkState.6 THEN //EC_LINK_STATE_PORT_C
	tempLookupSlaveDevState := CONCAT(tempLookupSlaveDevState, ' - ');
	tempLookupSlaveDevState := CONCAT(tempLookupSlaveDevState, 'Port 2');
END_IF

IF EcSlavesState[Slave].linkState.7 THEN //EC_LINK_STATE_PORT_D
	tempLookupSlaveDevState := CONCAT(tempLookupSlaveDevState, ' - ');
	tempLookupSlaveDevState := CONCAT(tempLookupSlaveDevState, 'Port 3');
END_IF

LookupSlaveDevState := tempLookupSlaveDevState;
END_METHOD

METHOD PRIVATE RaiseAlarmWithStringsAndFlags
VAR_INPUT
	Alarm	 : FB_TcAlarm; //! Alarm to be raised
	String_1 : STRING;
	String_2 : STRING;
	String_3 : STRING;
END_VAR
IF NOT Alarm.bRaised THEN
	F_RaiseAlarmWithStringsAndFlags(Alarm	  := Alarm,
									ErrorFlag := _Error,
									ErrorID	  := _ErrorID,
									String_1  := String_1,
									String_2  := String_2,
									String_3  := String_3);
END_IF
END_METHOD

METHOD PRIVATE RaiseWarningWithStringParameters
VAR_INPUT
	Warning	 : FB_TcAlarm; //! Alarm to be raised
	String_1 : STRING;
	String_2 : STRING;
	String_3 : STRING;
END_VAR
IF NOT Warning.bRaised THEN
	F_RaiseAlarmWithStringParameters(Alarm	  := Warning,
									 String_1 := String_1,
									 String_2 := String_2,
									 String_3 := String_3);
END_IF
END_METHOD

METHOD PRIVATE SlaveIsPartOfSyncUnit : BOOL
VAR_INPUT
	SlaveAddr : UINT;
	SyncUnit  : ST_SyncUnitInfo;
END_VAR

VAR_INST
	i : UDINT;
END_VAR
SlaveIsPartOfSyncUnit := FALSE;
FOR i := 1 TO Parameter_Diagnostic.ETHERCAT_MASTER_SYNC_UNIT_SLAVE_MAX DO
	IF SyncUnit.Slaves[i] = SlaveAddr THEN
		SlaveIsPartOfSyncUnit := TRUE;
		RETURN;
	END_IF
END_FOR
END_METHOD

METHOD FB_init : BOOL
VAR_INPUT
	bInitRetains	  : BOOL; // if TRUE, the retain variables are initialized (warm start / cold start)
	bInCopyCode		  : BOOL; // if TRUE, the instance afterwards gets moved into the copy code (online change)
	EtherCatSyncUnits : I_EtherCatSyncUnits;
END_VAR
IF EtherCatSyncUnits <> 0 THEN
	ipEtherCatSyncUnits := EtherCatSyncUnits;
END_IF
END_METHOD

//! @summary Provides interlocks for HMI control and updates HMI status information for this component
METHOD PROTECTED HMICommunication

//! @description This method is called cyclically by <c>CyclicLogic()</c>
SUPER^.HMICommunication();

// Device Info
EtherCatMaster_HMI.Config.DeviceInfo := _EtherCatMasterInfo;

// Status
EtherCatMaster_HMI.Status.EcSlavesState		  := EcSlavesState;
EtherCatMaster_HMI.Status.ConfiguredSlaveInfo := ConfiguredSlaveInfo;
EtherCatMaster_HMI.Status.EcSlaveTopologyInfo := EcSlaveTopologyInfo;
END_METHOD

//! @summary Basic component initialization logic
METHOD PROTECTED Initialize : BOOL;
VAR_INST
	InitializeSequence : UINT := 0;
	Size			   : UDINT;
	StartupTime		   : TON;
END_VAR

//! @description This method is called by <c>CyclicLogic()</c> as required
{analysis -19}
Initialize := FALSE;
IF NOT __ISVALIDREF(_EtherCatMasterInfo) THEN
	_Error := TRUE;
	Trace('Init Failed - EtherCatMasterInfo not set in EtherCat Master Component!');
END_IF

IF ipEtherCatSyncUnits = 0 THEN
	_Error := TRUE;
	Trace('Init Failed - EtherCatSyncUnits not set in constructor!');
END_IF

IF _Error THEN
	RETURN;
END_IF

IF _Simulate THEN
	Initialize := SUPER^.Initialize();
	RETURN;
END_IF

// Get all Slaves
GetConfiguredSlaves(sNetId				:= _EtherCatMasterInfo.AmsNetID,
					pArrEcConfSlaveInfo := ADR(ConfiguredSlaveInfo),
					cbBufLen			:= SIZEOF(ConfiguredSlaveInfo),
					tTimeout			:= T#1S);

// Init Sequence
CASE InitializeSequence OF
	(* Read Configured Slave Info Data *)
	0:
		GetConfiguredSlaves.bExecute := TRUE;
		IF GetConfiguredSlaves.bBusy THEN
			InitializeSequence := InitializeSequence + 10;
		END_IF

	10:
		IF NOT GetConfiguredSlaves.bBusy AND NOT GetConfiguredSlaves.bError THEN
			CfgSlaveCount := GetConfiguredSlaves.nSlaves;
			IF CfgSlaveCount > Parameter_Diagnostic.ETHERCAT_MASTER_SLAVE_MAX THEN
				Trace('Init Failed - Configured EtherCat Slave amount per master to small! Increase ETHERCAT_MASTER_SLAVE_MAX!');
			ELSE
				InitializeSequence := InitializeSequence + 10;
			END_IF
		END_IF

		IF GetConfiguredSlaves.bError THEN
			_Error := TRUE;
			Trace('Init Failed - Configured EtherCat Slaves could not be read!');
			InitializeSequence := 999;
		END_IF

	20: // Startup time for Ethercat Master	
		StartupTime(IN := TRUE, PT := Parameter_Diagnostic.ETHERCAT_MASTER_START_UP_TIME);
		IF StartupTime.Q THEN
			InitializeSequence := InitializeSequence + 10;
		END_IF

	30:
		Initialize := SUPER^.Initialize();
END_CASE
END_METHOD

METHOD PROTECTED MasterState
VAR_INST
	TypeError			 : BOOL;
	TypeWarning			 : BOOL;
	MasterDevStateString : STRING;
END_VAR
// Read Master state
EcGetMasterDevState(sNetId := _EtherCatMasterInfo.AmsNetID, tTimeout := T#1S, nDevState => MasterDevState);

// Sequence
CASE MasterSeq OF
	(* Wait for start *)
	0:
		EcGetMasterDevState.bExecute := FALSE;

	(* Read Master State*)
	10:
		EcGetMasterDevState.bExecute := TRUE;
		IF EcGetMasterDevState.bBusy THEN
			MasterSeq := MasterSeq + 10;
		END_IF

	20:
		IF NOT EcGetMasterDevState.bBusy AND NOT EcGetMasterDevState.bError THEN
			MasterSeq := MasterSeq + 10;
		END_IF

		IF EcGetMasterDevState.bError THEN
			MasterSeq := 999;
		END_IF

	(* Evaluate Master State *)
	30:
		MasterDevStateString := LookupMasterDevState(State := MasterDevState, TypeError => TypeError, TypeWarning => TypeWarning);
		IF MasterDevState <> 0 THEN
			IF TypeError THEN
				IF NOT MasterAlarms[E_EtherCatMaster.MasterError].bRaised THEN
					SUPER^.RaiseAlarmWithStrings(Alarm := MasterAlarms[E_EtherCatMaster.MasterError], String_1 := MasterDevStateString, String_2 := '');
				END_IF
			END_IF

			IF TypeWarning THEN
				IF NOT MasterAlarms[E_EtherCatMaster.MasterWarning].bRaised THEN
					SUPER^.RaiseEventWithStrings(Alarm := MasterAlarms[E_EtherCatMaster.MasterWarning], String_1 := MasterDevStateString, String_2 := '');
				END_IF
			END_IF

			_ErrorID := MasterDevState;
		END_IF

		MasterSeq := MasterSeq + 10;

	40:
		MasterSeq := 0;

	(* Sequence Error*)
	999:
		Trace('FB_Component_EtherCatMaster - Error get Master State Sequence!');
		MasterSeq := 0;
END_CASE
END_METHOD

METHOD PROTECTED SlaveState
VAR_INST
	BitMaskDiag	 : BYTE := 16#0F;
	ErrorSlave	 : BOOL;
	FaultedSlave : UDINT;
	SyncUnit	 : UDINT;

	// Sync Unit Diagnostic
	SlavesInSyncUnitPartA : STRING;
	SlavesInSyncUnitPartB : STRING;
END_VAR
{analysis -14}
{analysis -07}
{analysis -19}

// Get slave topology info
GetSlaveTopologyInfo(sNetId	  := _EtherCatMasterInfo.AmsNetID,
					 pAddrBuf := ADR(EcSlaveTopologyInfo),
					 cbBufLen := SIZEOF(EcSlaveTopologyInfo),
					 tTimeout := T#5S);

// Get all slave states
EcGetAllSlaveStates(sNetId	  := _EtherCatMasterInfo.AmsNetID,
					pStateBuf := ADR(EcSlavesState),
					cbBufLen  := SIZEOF(EcSlavesState),
					tTimeout  := T#5S);

// Sequence
CASE SlaveSeq OF
	(* Wait for start *)
	0:
		EcGetAllSlaveStates.bExecute  := FALSE;
		GetConfiguredSlaves.bExecute  := FALSE;
		GetSlaveTopologyInfo.bExecute := FALSE;

	(* Update Topology*)
	10:
		GetSlaveTopologyInfo.bExecute := TRUE;
		IF GetSlaveTopologyInfo.bBusy THEN
			SlaveSeq := SlaveSeq + 10;
		END_IF

	20:
		IF NOT GetSlaveTopologyInfo.bBusy AND NOT GetSlaveTopologyInfo.bError THEN
			SlaveSeq := SlaveSeq + 10;
		END_IF

		IF GetSlaveTopologyInfo.bError THEN
			SlaveSeq := 999;
		END_IF

	(* Update Sync Units*)
	30:
		ipEtherCatSyncUnits.Update();
		IF ipEtherCatSyncUnits.Busy THEN
			SlaveSeq := SlaveSeq + 10;
		END_IF

	40:
		IF NOT ipEtherCatSyncUnits.Busy AND NOT ipEtherCatSyncUnits.Error THEN
			// Get EtherCat Sync Units
			SyncUnits REF= ipEtherCatSyncUnits.SyncUnits;
			SlaveSeq  := SlaveSeq + 10;
		END_IF

		IF ipEtherCatSyncUnits.Error THEN
			SlaveSeq := 999;
		END_IF

	(* Read Slave States *)
	50:
		EcGetAllSlaveStates.bExecute := TRUE;
		IF EcGetAllSlaveStates.bBusy THEN
			SlaveSeq := SlaveSeq + 10;
		END_IF

	60:
		IF NOT EcGetAllSlaveStates.bBusy AND NOT EcGetAllSlaveStates.bError THEN
			SlaveCount := EcGetAllSlaveStates.nSlaves;
			SlaveSeq   := SlaveSeq + 10;
		END_IF

		IF EcGetAllSlaveStates.bError THEN
			SlaveSeq := 999;
		END_IF

	(* Evaluate Slave Error *)
	70:
		FOR FaultedSlave := 0 TO (CfgSlaveCount - 1) DO
			// Slave State
			IF (EcSlavesState[FaultedSlave].deviceState AND BitMaskDiag) <> EC_DEVICE_STATE_OP AND EcSlaveTopologyInfo[FaultedSlave].nStatusBits.4 = FALSE THEN
				IF EcSlavesState[FaultedSlave].deviceState.7 THEN // Slave is Disabled or hot connect- warning only
					THIS^.RaiseWarningWithStringParameters(Warning	:= SlaveWarnings[FaultedSlave],
														   String_1 := SlaveWarnings[FaultedSlave].ipSourceInfo.sName,
														   String_2 := LookupSlaveDevState(FaultedSlave),
														   String_3 := '');
				ELSE
					THIS^.RaiseAlarmWithStringsAndFlags(Alarm	 := SlaveErrors[FaultedSlave],
														String_1 := SlaveErrors[FaultedSlave].ipSourceInfo.sName,
														String_2 := LookupSlaveDevState(FaultedSlave),
														String_3 := '');

					ErrorSlave := TRUE;
				END_IF
			END_IF

			// Slave Linking Error
			IF (EcSlavesState[FaultedSlave].linkState AND BitMaskDiag) <> EC_LINK_STATE_OK AND EcSlaveTopologyInfo[FaultedSlave].nStatusBits.4 = FALSE THEN
				THIS^.RaiseAlarmWithStringsAndFlags(Alarm	 := SlaveErrors[FaultedSlave],
													String_1 := SlaveErrors[FaultedSlave].ipSourceInfo.sName,
													String_2 := LookupSlaveDevState(FaultedSlave),
													String_3 := '');
			END_IF

			// Raise related Sync Unit Alarm
			FOR SyncUnit := 1 TO Parameter_Diagnostic.ETHERCAT_MASTER_SYNC_UNIT_MAX DO
				IF SyncUnits[SyncUnit].Parent = THIS^.Name THEN
					IF SlaveIsPartOfSyncUnit(SlaveAddr := ConfiguredSlaveInfo[FaultedSlave].nAddr, SyncUnit := SyncUnits[SyncUnit]) AND SlaveErrors[FaultedSlave].bRaised OR SlaveWarnings[FaultedSlave].bRaised THEN
						THIS^.GetSyncUnitSlaveNames(SyncUnit := SyncUnits[SyncUnit], SlavesInSyncUnitPartA => SlavesInSyncUnitPartA, SlavesInSyncUnitPartB => SlavesInSyncUnitPartB);
						THIS^.RaiseWarningWithStringParameters(Warning	:= SyncUnitWarnings[SyncUnit],
															   String_1 := CONCAT(SyncUnits[SyncUnit].Parent, CONCAT(' - ', SyncUnits[SyncUnit].Name)),
															   String_2 := SlavesInSyncUnitPartA,
															   String_3 := SlavesInSyncUnitPartB);

						EXIT;
					END_IF
				END_IF
			END_FOR
		END_FOR

		SlaveSeq := SlaveSeq + 10;

	80:
		SlaveSeq := 0;

	(* Sequence Error*)
	999:
		Trace('FB_Component_EtherCatMaster - Error get Slave States Sequence!');
		SlaveSeq := 0;
END_CASE
END_METHOD

PROPERTY EtherCatMasterInfo : REFERENCE TO ST_DeviceInfo
SET
{analysis -21}
_EtherCatMasterInfo REF= EtherCatMasterInfo;
END_SET
END_PROPERTY

END_FUNCTION_BLOCK

// EtherCat Diagnostic/F_EtherCAT_VendorIDtoString
FUNCTION F_EtherCAT_VendorIDtoString : STRING
VAR_INPUT
	VendorId: UDINT;
END_VAR
VAR
END_VAR

CASE VendorId OF
	16#00000000:
		F_EtherCAT_VendorIDtoString := '';

	16#00000001:
		F_EtherCAT_VendorIDtoString := 'EtherCAT Technology Group';

	16#00000002:
		F_EtherCAT_VendorIDtoString := 'Beckhoff Automation GmbH';

	16#00000003:
		F_EtherCAT_VendorIDtoString := 'Scuola Superiore S. Anna';

	16#00000004:
		F_EtherCAT_VendorIDtoString := 'IXXAT Automation GmbH';

	16#00000005:
		F_EtherCAT_VendorIDtoString := 'Vector Informatik GmbH';

	16#00000006:
		F_EtherCAT_VendorIDtoString := 'KNESTEL Technologie & Elektronik GmbH';

	16#00000007:
		F_EtherCAT_VendorIDtoString := 'Janz Tec AG';

	16#00000009:
		F_EtherCAT_VendorIDtoString := 'A&C Institute of Shenyang University of Technology';

	16#0000000A:
		F_EtherCAT_VendorIDtoString := 'CMZ Sistemi Elettronici';

	16#0000000B:
		F_EtherCAT_VendorIDtoString := 'JSL Technology Co.,Ltd';

	16#0000000C:
		F_EtherCAT_VendorIDtoString := 'comemso GmbH';

	16#0000000D:
		F_EtherCAT_VendorIDtoString := 'Softing Industrial Automation GmbH';

	16#0000000E:
		F_EtherCAT_VendorIDtoString := 'MicroControl GmbH & Co. KG';

	16#0000000F:
		F_EtherCAT_VendorIDtoString := 'ESR Pollmeier GmbH';

	16#00000010:
		F_EtherCAT_VendorIDtoString := 'Beihang University, School of Mechanical Engineering & Automation';

	16#00000011:
		F_EtherCAT_VendorIDtoString := 'GKG Precision Machine Co., Ltd.';

	16#00000013:
		F_EtherCAT_VendorIDtoString := 'Fritz Kübler GmbH';

	16#00000014:
		F_EtherCAT_VendorIDtoString := 'KEB, Karl E. Brinkmann GmbH';

	16#00000015:
		F_EtherCAT_VendorIDtoString := 'AJINEXTEK Co. Ltd.';

	16#00000016:
		F_EtherCAT_VendorIDtoString := 'LTi DRiVES GmbH';

	16#00000017:
		F_EtherCAT_VendorIDtoString := 'esd electronic system design gmbh';

	16#00000018:
		F_EtherCAT_VendorIDtoString := 'M2I Corporation';

	16#0000001B:
		F_EtherCAT_VendorIDtoString := 'HMS Industrial Networks AB';

	16#0000001C:
		F_EtherCAT_VendorIDtoString := 'epis Automation GmbH & Co. KG';

	16#0000001D:
		F_EtherCAT_VendorIDtoString := 'Festo AG & Co. KG';

	16#00000021:
		F_EtherCAT_VendorIDtoString := 'WAGO Kontakttechnik GmbH & Co. KG';

	16#00000024:
		F_EtherCAT_VendorIDtoString := 'Bosch Rexroth AG';

	16#00000028:
		F_EtherCAT_VendorIDtoString := 'Moog GmbH';

	16#0000002A:
		F_EtherCAT_VendorIDtoString := 'HIGHYAG Lasertechnologie GmbH';

	16#00000034:
		F_EtherCAT_VendorIDtoString := 'port GmbH';

	16#00000039:
		F_EtherCAT_VendorIDtoString := 'Bürkert Werke GmbH';

	16#0000003B:
		F_EtherCAT_VendorIDtoString := 'Lenze SE';

	16#00000040:
		F_EtherCAT_VendorIDtoString := 'MTS Sensor Technologie GmbH & Co. KG';

	16#00000042:
		F_EtherCAT_VendorIDtoString := 'Tigris Electronic GmbH';

	16#00000044:
		F_EtherCAT_VendorIDtoString := 'Hilscher GmbH';

	16#0000004B:
		F_EtherCAT_VendorIDtoString := 'EVER s.n.c.';

	16#0000004F:
		F_EtherCAT_VendorIDtoString := 'Murrelektronik GmbH';

	16#00000051:
		F_EtherCAT_VendorIDtoString := 'PCS Power Converter Solutions GmbH';

	16#00000057:
		F_EtherCAT_VendorIDtoString := 'Komax AG';

	16#00000059:
		F_EtherCAT_VendorIDtoString := 'SEW-EURODRIVE GmbH & Co. KG';

	16#0000005D:
		F_EtherCAT_VendorIDtoString := 'Schleicher Electronic GmbH & Co. KG';

	16#00000062:
		F_EtherCAT_VendorIDtoString := 'Bachmann electronic GmbH';

	16#00000066:
		F_EtherCAT_VendorIDtoString := 'ROFIN-SINAR Laser GmbH';

	16#0000006A:
		F_EtherCAT_VendorIDtoString := 'KOLLMORGEN Corporation';

	(*16#0000006A: F_EtherCAT_VendorIDtoString :='KOLLMORGEN Europe GmbH';*)
	16#0000006B:
		F_EtherCAT_VendorIDtoString := 'Woodward SEG GmbH & Co. KG';

	16#0000006C:
		F_EtherCAT_VendorIDtoString := 'Bernecker + Rainer Industrie-Elektronik Ges.m.b.H';

	16#00000077:
		F_EtherCAT_VendorIDtoString := 'SLC Sautter Lift Components GmbH & Co. KG';

	16#00000082:
		F_EtherCAT_VendorIDtoString := 'Infranor SAS';

	16#00000083:
		F_EtherCAT_VendorIDtoString := 'OMRON Corporation';

	16#00000084:
		F_EtherCAT_VendorIDtoString := 'Phoenix Contact GmbH & Co. KG';

	16#0000008A:
		F_EtherCAT_VendorIDtoString := 'System S.p.A.';

	16#00000090:
		F_EtherCAT_VendorIDtoString := 'Vacon Plc';

	16#00000093:
		F_EtherCAT_VendorIDtoString := 'Gefran S.P.A.';

	16#00000099:
		F_EtherCAT_VendorIDtoString := 'SHENZHEN CO-TRUST TECHNOLOGY CO., LTD.';

	16#0000009A:
		F_EtherCAT_VendorIDtoString := 'Elmo Motion Control Ltd.';

	16#0000009C:
		F_EtherCAT_VendorIDtoString := 'Hans Turck GmbH & Co. KG';

	16#000000A0:
		F_EtherCAT_VendorIDtoString := 'Sontheim Industrie Elektronik GmbH';

	16#000000A2:
		F_EtherCAT_VendorIDtoString := 'HORIBA STEC, Co., Ltd.';

	16#000000A5:
		F_EtherCAT_VendorIDtoString := 'Hirschmann Automation and Control GmbH';

	16#000000AA:
		F_EtherCAT_VendorIDtoString := 'Bejing A&E Precision Machinery Co., Ltd.';

	16#000000AB:
		F_EtherCAT_VendorIDtoString := 'Copley Controls, a Division of Analogic Corporation';

	16#000000AD:
		F_EtherCAT_VendorIDtoString := 'Pepperl+Fuchs GmbH';

	16#000000AF:
		F_EtherCAT_VendorIDtoString := 'Johannes Hübner Fabrik elektrischer Maschinen GmbH';

	16#000000B3:
		F_EtherCAT_VendorIDtoString := 'Jetter AG';

	16#000000B7:
		F_EtherCAT_VendorIDtoString := 'ABB Oy Drives';

	16#000000B9:
		F_EtherCAT_VendorIDtoString := 'STÖBER ANTRIEBSTECHNIK GmbH & Co. KG';

	16#000000BC:
		F_EtherCAT_VendorIDtoString := 'AEC S.r.l.';

	16#000000BD:
		F_EtherCAT_VendorIDtoString := 'ADVANCED Motion Controls';

	16#000000BE:
		F_EtherCAT_VendorIDtoString := 'Bloom Energy (India) Private Limited';

	16#000000C5:
		F_EtherCAT_VendorIDtoString := 'Comdel, Inc.';

	16#000000CE:
		F_EtherCAT_VendorIDtoString := 'Mitsubishi Electric India Pvt. Ltd.';

	16#000000D5:
		F_EtherCAT_VendorIDtoString := 'BONFIGLIOLI VECTRON GmbH';

	16#000000D9:
		F_EtherCAT_VendorIDtoString := 'Phase Motion Control SpA';

	16#000000DA:
		F_EtherCAT_VendorIDtoString := 'Diener Automation GmbH & Co. KG';

	16#000000E2:
		F_EtherCAT_VendorIDtoString := 'plating electronic GmbH';

	16#000000E4:
		F_EtherCAT_VendorIDtoString := 'Metronix Messgeräte und Elektronik GmbH';

	16#000000E9:
		F_EtherCAT_VendorIDtoString := 'Ascon S.p.A.';

	16#000000EA:
		F_EtherCAT_VendorIDtoString := 'ESAB-ATAS GmbH';

	16#000000EB:
		F_EtherCAT_VendorIDtoString := 'Elektrobit Automotive GmbH';

	16#000000EC:
		F_EtherCAT_VendorIDtoString := 'Baumer IVO GmbH & Co. KG';

	16#000000F1:
		F_EtherCAT_VendorIDtoString := 'McLaren Group Limited';

	16#000000F2:
		F_EtherCAT_VendorIDtoString := 'Guangdong University of Technology';

	16#000000F4:
		F_EtherCAT_VendorIDtoString := 'Atos SpA';

	16#000000F5:
		F_EtherCAT_VendorIDtoString := 'Giant Magellan Telescope Corporation';

	16#000000F9:
		F_EtherCAT_VendorIDtoString := 'Control Techniques Ltd.';

	16#000000FB:
		F_EtherCAT_VendorIDtoString := 'maxon motor ag';

	16#000000FE:
		F_EtherCAT_VendorIDtoString := 'Precitec KG';

	16#000000FF:
		F_EtherCAT_VendorIDtoString := 'South China University of Technology';

	16#00000101:
		F_EtherCAT_VendorIDtoString := 'ISAC Srl.';

	16#00000104:
		F_EtherCAT_VendorIDtoString := 'LMD GmbH & Co. KG aA';

	16#00000105:
		F_EtherCAT_VendorIDtoString := 'KEBA AG';

	16#0000010A:
		F_EtherCAT_VendorIDtoString := 'WITTENSTEIN motion control GmbH';

	16#0000010D:
		F_EtherCAT_VendorIDtoString := 'TWK-Elektronik GmbH';

	16#0000010F:
		F_EtherCAT_VendorIDtoString := 'PSA Elettronica di F. Grifa';

	16#00000111:
		F_EtherCAT_VendorIDtoString := 'HEITEC AG';

	(*16#00000114: F_EtherCAT_VendorIDtoString :='SMC European Technical Centre';*)
	16#00000114:
		F_EtherCAT_VendorIDtoString := 'SMC Corporation';

	(*16#00000114: F_EtherCAT_VendorIDtoString :='SMC Corporation of America';*)
	16#00000116:
		F_EtherCAT_VendorIDtoString := 'Eckelmann AG';

	16#00000117:
		F_EtherCAT_VendorIDtoString := 'JVL Industri Elektronik A/S';

	16#0000011D:
		F_EtherCAT_VendorIDtoString := 'Hottinger Baldwin Messtechnik GmbH';

	16#00000121:
		F_EtherCAT_VendorIDtoString := 'Leuze electronic GmbH + Co. KG';

	16#00000123:
		F_EtherCAT_VendorIDtoString := 'WEG Equipamentos Elétricos S.A.';

	16#00000126:
		F_EtherCAT_VendorIDtoString := 'JUMO GmbH & Co. KG';

	16#00000129:
		F_EtherCAT_VendorIDtoString := 'HSD S.p.A';

	16#0000012E:
		F_EtherCAT_VendorIDtoString := 'Lika Electronic Srl';

	16#0000012F:
		F_EtherCAT_VendorIDtoString := 'CSM GmbH';

	16#00000137:
		F_EtherCAT_VendorIDtoString := 'Fenwal Controls of Japan,Ltd.';

	16#00000144:
		F_EtherCAT_VendorIDtoString := 'TECNOLOGIX Srl';

	16#00000146:
		F_EtherCAT_VendorIDtoString := 'LPKF SolarQuipment GmbH';

	16#00000147:
		F_EtherCAT_VendorIDtoString := 'Dr. Fritz Faulhaber GmbH & Co. KG';

	16#0000014A:
		F_EtherCAT_VendorIDtoString := 'imc Messysteme GmbH';

	16#0000015A:
		F_EtherCAT_VendorIDtoString := 'Baumüller Nürnberg GmbH';

	16#00000166:
		F_EtherCAT_VendorIDtoString := 'Metso Automation Oy';

	16#00000168:
		F_EtherCAT_VendorIDtoString := 'Shanghai AMP&MOONS Automation Co., Ltd.';

	16#0000016D:
		F_EtherCAT_VendorIDtoString := 'COMSOFT GmbH';

	16#00000171:
		F_EtherCAT_VendorIDtoString := 'Prima Electro S.p.A.';

	16#0000017A:
		F_EtherCAT_VendorIDtoString := 'Pneumax S.p.A.';

	16#0000017F:
		F_EtherCAT_VendorIDtoString := 'R.T.A. S.r.l.';

	16#00000190:
		F_EtherCAT_VendorIDtoString := 'Promess Incorporated';

	16#00000191:
		F_EtherCAT_VendorIDtoString := 'PROMESS Gesellschaft für Montage- und Prüfsysteme mbH';

	16#0000019D:
		F_EtherCAT_VendorIDtoString := 'Deutschmann Automation GmbH & Co. KG';

	16#0000019E:
		F_EtherCAT_VendorIDtoString := 'Golden A/S';

	16#000001A1:
		F_EtherCAT_VendorIDtoString := 'Brunner Elektronik AG';

	16#000001A3:
		F_EtherCAT_VendorIDtoString := 'TECHNOSOFT S.A.';

	16#000001B4:
		F_EtherCAT_VendorIDtoString := 'Peyer Engineering';

	16#000001B5:
		F_EtherCAT_VendorIDtoString := 'Robox S.P.A.';

	16#000001B9:
		F_EtherCAT_VendorIDtoString := 'Sanyo Denki Co., Ltd.';

	16#000001C0:
		F_EtherCAT_VendorIDtoString := 'Kobe Steel, Ltd.';

	16#000001C4:
		F_EtherCAT_VendorIDtoString := 'Regatron AG';

	16#000001DD:
		F_EtherCAT_VendorIDtoString := 'Delta Electronics, Inc.';

	16#000001DF:
		F_EtherCAT_VendorIDtoString := 'Xeikon N.V. - Xeikon Manufacturing and R&D Center';

	16#000001E1:
		F_EtherCAT_VendorIDtoString := 'Numatics Inc.';

	16#000001EB:
		F_EtherCAT_VendorIDtoString := 'AMK Arnold Müller GmbH & Co. KG';

	16#000001F9:
		F_EtherCAT_VendorIDtoString := 'National Instruments Corporation';

	16#000001FC:
		F_EtherCAT_VendorIDtoString := 'Fernsteuergeräte Kurt Oelsch GmbH';

	16#000001FD:
		F_EtherCAT_VendorIDtoString := 'INA - Drives & Mechatronics GmbH & Co.oHG';

	16#000001FE:
		F_EtherCAT_VendorIDtoString := 'PRÜFTECHNIK NDT GmbH';

	16#00000205:
		F_EtherCAT_VendorIDtoString := 'TDE MACNO S.p.A.';

	16#00000207:
		F_EtherCAT_VendorIDtoString := 'esitron-electronic GmbH';

	16#00000219:
		F_EtherCAT_VendorIDtoString := 'Real Time Automation, Inc.';

	16#00000223:
		F_EtherCAT_VendorIDtoString := 'Systeme Helmholz GmbH';

	16#00000225:
		F_EtherCAT_VendorIDtoString := 'Pantec Engineering AG';

	16#0000022B:
		F_EtherCAT_VendorIDtoString := 'VIPA Gesellschaft für Visualisierung und Prozessautomatisierung mbH';

	16#00000230:
		F_EtherCAT_VendorIDtoString := 'Weidmüller Interface GmbH & Co. KG';

	16#0000023A:
		F_EtherCAT_VendorIDtoString := 'ABB Automation Products GmbH';

	16#0000023B:
		F_EtherCAT_VendorIDtoString := 'Berghof Automationstechnik GmbH';

	16#0000023D:
		F_EtherCAT_VendorIDtoString := 'Sensor-Technik Wiedemann GmbH';

	16#00000240:
		F_EtherCAT_VendorIDtoString := 'Spezialantriebstechnik GmbH';

	16#00000247:
		F_EtherCAT_VendorIDtoString := 'Harmonic Drive LLC';

	16#0000024F:
		F_EtherCAT_VendorIDtoString := 'Stotz Feinmesstechnik GmbH';

	16#00000257:
		F_EtherCAT_VendorIDtoString := 'Dunkermotoren GmbH';

	16#0000025E:
		F_EtherCAT_VendorIDtoString := 'Fuji Electric Co., Ltd.';

	16#00000260:
		F_EtherCAT_VendorIDtoString := 'TRUMPF Hüttinger GmbH + Co. KG';

	16#0000026C:
		F_EtherCAT_VendorIDtoString := 'Nanotec Electronic GmbH & Co. KG';

	16#00000279:
		F_EtherCAT_VendorIDtoString := 'ISH Ingenieursozietät GmbH';

	16#00000283:
		F_EtherCAT_VendorIDtoString := 'Roche Diagnostics AG';

	16#00000284:
		F_EtherCAT_VendorIDtoString := 'Toshiba Schneider Inverter Corporation';

	16#00000285:
		F_EtherCAT_VendorIDtoString := 'Bihl-Wiedemann GmbH';

	16#00000286:
		F_EtherCAT_VendorIDtoString := 'TRINAMIC Motion Control GmbH & Co. KG';

	16#00000289:
		F_EtherCAT_VendorIDtoString := 'HDT Srl';

	16#00000292:
		F_EtherCAT_VendorIDtoString := 'Horner APG LLC';

	16#00000296:
		F_EtherCAT_VendorIDtoString := 'Performance Motion Devices, Inc.';

	16#0000029C:
		F_EtherCAT_VendorIDtoString := 'INGENIA-CAT, S.L.';

	16#0000029D:
		F_EtherCAT_VendorIDtoString := 'CREVIS Co., Ltd.';

	16#000002B9:
		F_EtherCAT_VendorIDtoString := 'Advanced Energy Industries, Inc.';

	16#000002BE:
		F_EtherCAT_VendorIDtoString := 'ORIENTAL MOTOR CO., LTD.';

	16#000002C1:
		F_EtherCAT_VendorIDtoString := 'Fronius International GmbH';

	16#000002D0:
		F_EtherCAT_VendorIDtoString := 'THK Co., Ltd.';

	16#000002D8:
		F_EtherCAT_VendorIDtoString := 'halstrup-walcher GmbH';

	16#000002D9:
		F_EtherCAT_VendorIDtoString := 'Walcher Meßtechnik GmbH';

	16#000002DE:
		F_EtherCAT_VendorIDtoString := 'Trio Motion Technology Ltd.';

	16#000002E1:
		F_EtherCAT_VendorIDtoString := 'Servotronix Motion Control Ltd.';

	16#000002EB:
		F_EtherCAT_VendorIDtoString := 'Analytica GmbH';

	16#000002EE:
		F_EtherCAT_VendorIDtoString := 'Metal Work S.p.A';

	16#00000302:
		F_EtherCAT_VendorIDtoString := 'Digitronic Automationsanlagen GmbH';

	16#0000030C:
		F_EtherCAT_VendorIDtoString := 'LAM Technologies S.a.S.';

	16#0000030E:
		F_EtherCAT_VendorIDtoString := 'IEP Ingenieurbüro für Echtzeitprogrammierung GmbH';

	16#00000311:
		F_EtherCAT_VendorIDtoString := 'Mikrap AG';

	16#00000312:
		F_EtherCAT_VendorIDtoString := 'A-KYUNG Motion Inc.';

	16#00000317:
		F_EtherCAT_VendorIDtoString := 'TOFLO CORPORATION';

	16#00000318:
		F_EtherCAT_VendorIDtoString := 'AXIS CORPORATION';

	16#00000321:
		F_EtherCAT_VendorIDtoString := '3S - Smart Software Solutions GmbH';

	16#00000326:
		F_EtherCAT_VendorIDtoString := 'GE Intelligent Plattforms';

	16#00000331:
		F_EtherCAT_VendorIDtoString := 'SHANGHAI SANY SCIENCE & TECHNOLOGY CO., LTD';

	16#00000334:
		F_EtherCAT_VendorIDtoString := 'CYBELEC S.A.';

	16#00000337:
		F_EtherCAT_VendorIDtoString := 'KOSTAL Industrie Elektrik GmbH';

	16#0000033D:
		F_EtherCAT_VendorIDtoString := 'RS Automation Co., Ltd.';

	16#00000343:
		F_EtherCAT_VendorIDtoString := 'K.C.Tech CO.,LTD.';

	16#00000344:
		F_EtherCAT_VendorIDtoString := 'Exlar Corporation';

	16#0000034D:
		F_EtherCAT_VendorIDtoString := 'Schaefer Elektronik GmbH';

	16#0000034E:
		F_EtherCAT_VendorIDtoString := 'Infineon Technologies AG';

	16#00000367:
		F_EtherCAT_VendorIDtoString := 'Novatech-Group Ltd.';

	16#00000384:
		F_EtherCAT_VendorIDtoString := 'MKS Denmark ApS';

	16#000003AE:
		F_EtherCAT_VendorIDtoString := 'HanYang System';

	16#000003DB:
		F_EtherCAT_VendorIDtoString := 'Baldor UK Ltd';

	16#000004D2:
		F_EtherCAT_VendorIDtoString := 'Noda Radio Frequency Technologies Co., Ltd.';

	16#00000500:
		F_EtherCAT_VendorIDtoString := 'Speciaal Machinefabriek Ketels v.o.f.';

	16#00000501:
		F_EtherCAT_VendorIDtoString := 'Beck IPC GmbH';

	16#00000502:
		F_EtherCAT_VendorIDtoString := 'ETAS GmbH';

	16#00000504:
		F_EtherCAT_VendorIDtoString := 'PHYTEC Messtechnik GmbH';

	16#00000505:
		F_EtherCAT_VendorIDtoString := 'ANCA Motion Pty. Ltd';

	16#00000506:
		F_EtherCAT_VendorIDtoString := 'Fachhochschule Köln';

	16#00000508:
		F_EtherCAT_VendorIDtoString := 'Nuvation Research Corporation';

	16#00000509:
		F_EtherCAT_VendorIDtoString := 'TR-Electronic';

	16#0000050A:
		F_EtherCAT_VendorIDtoString := 'Gantner Instruments GmbH';

	16#0000050B:
		F_EtherCAT_VendorIDtoString := 'MKS Instruments';

	16#0000050C:
		F_EtherCAT_VendorIDtoString := 'ABB AB';

	(*16#0000050C: F_EtherCAT_VendorIDtoString :='ABB Engineering (Shanghai) Ltd.';*)
	16#0000050D:
		F_EtherCAT_VendorIDtoString := 'Unitro-Fleischmann';

	16#0000050E:
		F_EtherCAT_VendorIDtoString := 'zub machine control AG';

	16#0000050F:
		F_EtherCAT_VendorIDtoString := 'dSPACE GmbH';

	16#00000511:
		F_EtherCAT_VendorIDtoString := 'Samsung Heavy Industries';

	16#00000512:
		F_EtherCAT_VendorIDtoString := 'BCE Elektronik GmbH';

	16#00000513:
		F_EtherCAT_VendorIDtoString := 'Jäger Computergesteuerte Messtechnik GmbH';

	16#00000514:
		F_EtherCAT_VendorIDtoString := 'TETRA Gesellschaft für Sensorik, Robotik und Automation mbH';

	16#00000515:
		F_EtherCAT_VendorIDtoString := 'Justek Inc.';

	16#00000516:
		F_EtherCAT_VendorIDtoString := 'Baumer Thalheim GmbH & Co. KG';

	16#00000517:
		F_EtherCAT_VendorIDtoString := 'Elin EBG Traction GmbH';

	16#00000518:
		F_EtherCAT_VendorIDtoString := 'Meka Robotics';

	16#00000519:
		F_EtherCAT_VendorIDtoString := 'Altera Japan Ltd.';

	16#0000051A:
		F_EtherCAT_VendorIDtoString := 'EBV Elektronik GmbH & Co KG';

	16#0000051B:
		F_EtherCAT_VendorIDtoString := 'Ingenieurgemeinschaft IgH';

	16#0000051C:
		F_EtherCAT_VendorIDtoString := 'IAV GmbH';

	16#0000051D:
		F_EtherCAT_VendorIDtoString := 'Hitachi Industrial Equipment Systems';

	16#0000051E:
		F_EtherCAT_VendorIDtoString := 'TenAsys Corp.';

	16#0000051F:
		F_EtherCAT_VendorIDtoString := 'PONDis AG';

	16#00000520:
		F_EtherCAT_VendorIDtoString := 'Moog Italiana S.r.l.';

	16#00000522:
		F_EtherCAT_VendorIDtoString := 'Wallner Automation';

	16#00000523:
		F_EtherCAT_VendorIDtoString := 'AVL List GmbH';

	16#00000524:
		F_EtherCAT_VendorIDtoString := 'RITTER-Elektronik GmbH';

	16#00000527:
		F_EtherCAT_VendorIDtoString := 'Zwick GmbH & Co. KG';

	16#00000528:
		F_EtherCAT_VendorIDtoString := 'dresden elektronik ingenieurtechnik gmbh';

	16#00000529:
		F_EtherCAT_VendorIDtoString := 'Tokyo Keiso Co., Ltd.';

	16#0000052C:
		F_EtherCAT_VendorIDtoString := 'Philips Healthcare (CT Division)';

	16#0000052D:
		F_EtherCAT_VendorIDtoString := 'Chess B.V.';

	16#0000052E:
		F_EtherCAT_VendorIDtoString := 'NCT kft';

	16#0000052F:
		F_EtherCAT_VendorIDtoString := 'Anywire Corporation';

	16#00000530:
		F_EtherCAT_VendorIDtoString := 'Shadow Robot Company Ltd.';

	16#00000531:
		F_EtherCAT_VendorIDtoString := 'FeCon GmbH';

	16#00000532:
		F_EtherCAT_VendorIDtoString := 'FH Südwestfalen, Fachbereich Elektrische Energietechnik';

	16#00000533:
		F_EtherCAT_VendorIDtoString := 'add2 Ldt';

	16#00000534:
		F_EtherCAT_VendorIDtoString := 'ARM Automation, Inc.';

	16#00000537:
		F_EtherCAT_VendorIDtoString := 'KNAPP AG';

	16#00000538:
		F_EtherCAT_VendorIDtoString := 'Getriebebau NORD GmbH & Co. KG';

	16#00000539:
		F_EtherCAT_VendorIDtoString := 'Yaskawa Electric Corporation';

	16#0000053A:
		F_EtherCAT_VendorIDtoString := 'Oki Information Systems Co., Ltd.';

	16#0000053B:
		F_EtherCAT_VendorIDtoString := 'Takasaki Kyoudou Computing Center Co.';

	16#0000053C:
		F_EtherCAT_VendorIDtoString := 'NITTETSU ELEX Co., Ltd.';

	16#0000053E:
		F_EtherCAT_VendorIDtoString := 'Unjo AB';

	16#0000053F:
		F_EtherCAT_VendorIDtoString := 'EADS Deutschland GmbH';

	16#00000540:
		F_EtherCAT_VendorIDtoString := 'ACS Motion Control Ltd.';

	16#00000541:
		F_EtherCAT_VendorIDtoString := 'KEYENCE Corporation';

	16#00000542:
		F_EtherCAT_VendorIDtoString := 'MEFI s.r.o.';

	16#00000543:
		F_EtherCAT_VendorIDtoString := 'm-u-t AG Messgeräte für Medizin- und Umwelttechnik';

	16#00000544:
		F_EtherCAT_VendorIDtoString := 'Universität Stuttgart, Institut ISW';

	16#00000545:
		F_EtherCAT_VendorIDtoString := 'ELSENA, Inc.';

	16#00000546:
		F_EtherCAT_VendorIDtoString := 'BE Semiconductor Industries N.V.';

	16#00000547:
		F_EtherCAT_VendorIDtoString := 'Hauni LNI Electronics S.A.';

	16#00000548:
		F_EtherCAT_VendorIDtoString := 'ETEL S.A.';

	16#00000549:
		F_EtherCAT_VendorIDtoString := 'VAT Vakuumventile AG';

	16#0000054A:
		F_EtherCAT_VendorIDtoString := 'LayTec AG';

	16#0000054B:
		F_EtherCAT_VendorIDtoString := 'NUM AG';

	16#0000054C:
		F_EtherCAT_VendorIDtoString := 'Hauni Maschinenbau AG';

	16#0000054D:
		F_EtherCAT_VendorIDtoString := 'Exatronic, Engenharia Electrónica, Lda';

	16#0000054E:
		F_EtherCAT_VendorIDtoString := 'Chinese Academy of Sciences, Institute of Intelligent Machines';

	16#0000054F:
		F_EtherCAT_VendorIDtoString := 'Eindhoven University of Technology';

	16#00000550:
		F_EtherCAT_VendorIDtoString := 'Scansonic MI GmbH';

	16#00000551:
		F_EtherCAT_VendorIDtoString := 'Shanghai Sodick Software Co., Ltd.';

	16#00000552:
		F_EtherCAT_VendorIDtoString := 'CHUO ELECTRONICS CO., LTD';

	16#00000553:
		F_EtherCAT_VendorIDtoString := 'Agie Charmilles SA';

	16#00000554:
		F_EtherCAT_VendorIDtoString := 'miControl GmbH';

	16#00000555:
		F_EtherCAT_VendorIDtoString := 'Haute Ecole dIngénierie et de Gestion du Canton de Vaud';

	16#00000557:
		F_EtherCAT_VendorIDtoString := 'Jenny Science AG';

	16#00000558:
		F_EtherCAT_VendorIDtoString := 'Industrial Control Communications, Inc.';

	16#0000055A:
		F_EtherCAT_VendorIDtoString := '?KD ELEKTROTECHNIKA, a.s.';

	16#0000055B:
		F_EtherCAT_VendorIDtoString := 'QEM S.r.l.';

	16#0000055C:
		F_EtherCAT_VendorIDtoString := 'Simatex AG';

	16#0000055D:
		F_EtherCAT_VendorIDtoString := 'Kithara Software GmbH';

	16#0000055E:
		F_EtherCAT_VendorIDtoString := 'GE Energy Power Conversion GmbH';

	16#0000055F:
		F_EtherCAT_VendorIDtoString := 'ARA apparatenfabriek b.v.';

	16#00000560:
		F_EtherCAT_VendorIDtoString := 'Tata Consultancy Services Ltd.';

	16#00000561:
		F_EtherCAT_VendorIDtoString := 'Harmonic Drive Systems Inc.';

	16#00000562:
		F_EtherCAT_VendorIDtoString := 'Tiab Limited';

	16#00000563:
		F_EtherCAT_VendorIDtoString := 'RKC INSTRUMENT INC.';

	16#00000564:
		F_EtherCAT_VendorIDtoString := 'Switched Reluctance Drives Ltd.';

	16#00000566:
		F_EtherCAT_VendorIDtoString := 'Avnet Electronics Marketing';

	16#00000567:
		F_EtherCAT_VendorIDtoString := 'ABB AB';

	16#00000568:
		F_EtherCAT_VendorIDtoString := 'Yamaha Motor Co., Ltd.';

	16#00000569:
		F_EtherCAT_VendorIDtoString := 'KUNBUS GmbH';

	16#0000056A:
		F_EtherCAT_VendorIDtoString := 'ACD Antriebstechnik GmbH';

	16#0000056B:
		F_EtherCAT_VendorIDtoString := 'Bronkhorst High-Tech B.V.';

	16#0000056C:
		F_EtherCAT_VendorIDtoString := 'K.MECS Co., Ltd.';

	16#0000056D:
		F_EtherCAT_VendorIDtoString := 'Ampegon AG';

	16#0000056E:
		F_EtherCAT_VendorIDtoString := 'UFG Elettronica s.r.l.';

	16#0000056F:
		F_EtherCAT_VendorIDtoString := 'Xilinx Ireland';

	16#00000570:
		F_EtherCAT_VendorIDtoString := 'ABB AB';

	16#00000571:
		F_EtherCAT_VendorIDtoString := 'Servoland Corporation';

	16#00000572:
		F_EtherCAT_VendorIDtoString := 'Hivertec, Inc.';

	16#00000573:
		F_EtherCAT_VendorIDtoString := 'Mesa Electronics';

	16#00000574:
		F_EtherCAT_VendorIDtoString := 'OMICRON electronics GmbH';

	16#00000575:
		F_EtherCAT_VendorIDtoString := 'Fike Europe B.v.b.a.';

	16#00000576:
		F_EtherCAT_VendorIDtoString := 'ROPEX Industrie-Elektronik GmbH';

	16#00000577:
		F_EtherCAT_VendorIDtoString := 'TLU - Thüringer Leistungselektronik Union GmbH';

	16#00000579:
		F_EtherCAT_VendorIDtoString := 'Prodrive B.V.';

	16#0000057A:
		F_EtherCAT_VendorIDtoString := 'miho Inspektionssysteme GmbH';

	16#0000057B:
		F_EtherCAT_VendorIDtoString := 'Tokyo Electron Device Limited';

	16#0000057C:
		F_EtherCAT_VendorIDtoString := 'LINTEC CO., LTD.';

	16#0000057D:
		F_EtherCAT_VendorIDtoString := 'Symplex Vision Systems GmbH';

	16#0000057E:
		F_EtherCAT_VendorIDtoString := 'Seiko Epson Corporation';

	16#0000057F:
		F_EtherCAT_VendorIDtoString := 'ZINSER Schweißtechnik GmbH';

	16#00000580:
		F_EtherCAT_VendorIDtoString := 'abk-technology GmbH';

	16#00000581:
		F_EtherCAT_VendorIDtoString := 'SUS Corporation';

	16#00000582:
		F_EtherCAT_VendorIDtoString := 'TRsystems GmbH';

	16#00000583:
		F_EtherCAT_VendorIDtoString := 'Harmonic Drive AG';

	16#00000584:
		F_EtherCAT_VendorIDtoString := 'Stäubli Faverges SCA';

	16#00000585:
		F_EtherCAT_VendorIDtoString := 'ScienLab electronic systems GmbH';

	16#00000586:
		F_EtherCAT_VendorIDtoString := 'DETO Mechatronic GmbH';

	16#00000587:
		F_EtherCAT_VendorIDtoString := 'FUJISOFT Incorporated';

	16#00000588:
		F_EtherCAT_VendorIDtoString := 'IAI Corporation';

	16#00000589:
		F_EtherCAT_VendorIDtoString := 'PromAvtomatika';

	16#0000058A:
		F_EtherCAT_VendorIDtoString := 'Kistler Instrumente AG';

	16#0000058B:
		F_EtherCAT_VendorIDtoString := 'LAUDA DR. R. WOBSER GmbH & Co. KG';

	16#0000058C:
		F_EtherCAT_VendorIDtoString := 'Schweitzer Engineering Laboratories, Inc.';

	16#0000058D:
		F_EtherCAT_VendorIDtoString := 'Vital Systems Inc.';

	16#0000058E:
		F_EtherCAT_VendorIDtoString := 'Mutracx B.V.';

	16#0000058F:
		F_EtherCAT_VendorIDtoString := 'Algo System Co., Ltd.';

	16#00000590:
		F_EtherCAT_VendorIDtoString := 'Mühlbauer AG';

	16#00000591:
		F_EtherCAT_VendorIDtoString := 'DETO Mechatronic GmbH';

	16#00000592:
		F_EtherCAT_VendorIDtoString := 'Sealevel Systems, Inc.';

	16#00000593:
		F_EtherCAT_VendorIDtoString := 'igm Robotersysteme AG';

	16#00000594:
		F_EtherCAT_VendorIDtoString := 'WITTENSTEIN electronics GmbH';

	16#00000595:
		F_EtherCAT_VendorIDtoString := 'ZBE Inc.';

	16#00000597:
		F_EtherCAT_VendorIDtoString := 'Fraunhofer IOSB-INA Kompetenzzentrum Industrial Automation';

	16#00000598:
		F_EtherCAT_VendorIDtoString := 'SKF Magnetic Bearings';

	16#00000599:
		F_EtherCAT_VendorIDtoString := 'Galil Motion Control Inc.';

	16#0000059A:
		F_EtherCAT_VendorIDtoString := 'IHI Corporation';

	16#0000059B:
		F_EtherCAT_VendorIDtoString := 'wenglor sensoric gmbh';

	16#0000059C:
		F_EtherCAT_VendorIDtoString := 'Ingeteam Technology S.A.';

	16#0000059D:
		F_EtherCAT_VendorIDtoString := 'Texas Instruments Incorporated';

	16#0000059E:
		F_EtherCAT_VendorIDtoString := 'Micro-Vu Corporation';

	16#0000059F:
		F_EtherCAT_VendorIDtoString := 'oehri electronic ag';

	16#000005A0:
		F_EtherCAT_VendorIDtoString := 'Triphase N.V.';

	16#00000600:
		F_EtherCAT_VendorIDtoString := 'Nagano Oki Electric Co., Ltd.';

	16#00000601:
		F_EtherCAT_VendorIDtoString := 'Condalo GmbH';

	16#00000602:
		F_EtherCAT_VendorIDtoString := 'Brooks Instrument, LLC';

	16#00000604:
		F_EtherCAT_VendorIDtoString := 'Leica Geosystems AG';

	16#00000605:
		F_EtherCAT_VendorIDtoString := 'Nabtesco Corporation';

	16#00000606:
		F_EtherCAT_VendorIDtoString := 'BP&M Representações e Consultoria LTDA';

	16#00000607:
		F_EtherCAT_VendorIDtoString := 'MICRO-EPSILON Optronic GmbH';

	16#00000608:
		F_EtherCAT_VendorIDtoString := 'Diamond Technologies, Inc.';

	16#0000060A:
		F_EtherCAT_VendorIDtoString := 'Estun Industrial Automation Co., Ltd.';

	16#0000060B:
		F_EtherCAT_VendorIDtoString := 'IMS Messsysteme GmbH';

	16#0000060C:
		F_EtherCAT_VendorIDtoString := 'M-System Co., Ltd.';

	16#0000060D:
		F_EtherCAT_VendorIDtoString := 'Ferrotec (USA) Corporation - Temescal Division';

	16#0000060E:
		F_EtherCAT_VendorIDtoString := 'SICK IVP AB';

	16#00000610:
		F_EtherCAT_VendorIDtoString := 'SINFONIA TECHNOLOGY CO., LTD.';

	16#00000611:
		F_EtherCAT_VendorIDtoString := 'Pfeiffer Vacuum GmbH';

	16#00000612:
		F_EtherCAT_VendorIDtoString := 'Froude Hofmann Limited';

	16#00000613:
		F_EtherCAT_VendorIDtoString := 'SABO Elektronik GmbH';

	16#00000615:
		F_EtherCAT_VendorIDtoString := 'Bystronic Laser AG';

	16#00000616:
		F_EtherCAT_VendorIDtoString := 'Shanghai Kinway Technologies, Inc.';

	16#00000618:
		F_EtherCAT_VendorIDtoString := 'LumaSense Technologies GmbH';

	16#00000619:
		F_EtherCAT_VendorIDtoString := 'BBH Products GmbH';

	16#0000061A:
		F_EtherCAT_VendorIDtoString := 'Hecht Automatisierungs-Systeme GmbH';

	16#0000061B:
		F_EtherCAT_VendorIDtoString := 'Xelmo AB';

	16#0000061C:
		F_EtherCAT_VendorIDtoString := 'Carl Zeiss Industrielle Messtechnik GmbH';

	16#0000061D:
		F_EtherCAT_VendorIDtoString := 'University of Genova, Faculty of Engineering';

	16#0000061E:
		F_EtherCAT_VendorIDtoString := 'Master Automation Group Oy';

	16#0000061F:
		F_EtherCAT_VendorIDtoString := 'Sankyo Seisakusho Co.';

	16#00000620:
		F_EtherCAT_VendorIDtoString := 'ATV-Elektronik Ges.m.b.H.';

	16#00000621:
		F_EtherCAT_VendorIDtoString := 'Panasonic Industrial Devices SUNX Co., Ltd.';

	16#00000622:
		F_EtherCAT_VendorIDtoString := 'ifm electronic gmbh';

	16#00000623:
		F_EtherCAT_VendorIDtoString := 'Fisher Technical Services Inc.';

	16#00000624:
		F_EtherCAT_VendorIDtoString := 'SCLE SFE';

	16#00000625:
		F_EtherCAT_VendorIDtoString := 'HIGEN Motor Co., Ltd.';

	16#00000626:
		F_EtherCAT_VendorIDtoString := 'Baumer hhs GmbH';

	16#00000627:
		F_EtherCAT_VendorIDtoString := 'Moog Inc.';

	16#00000628:
		F_EtherCAT_VendorIDtoString := 'XIOS Hogeschool Limburg, Department N-Technology';

	16#00000629:
		F_EtherCAT_VendorIDtoString := 'Azbil Corporation';

	16#0000062A:
		F_EtherCAT_VendorIDtoString := 'Delta Tau Data Systems, Inc.';

	16#0000062B:
		F_EtherCAT_VendorIDtoString := 'Heraeus Electro-Nite International N.V.';

	16#0000062C:
		F_EtherCAT_VendorIDtoString := 'ESW GmbH';

	16#0000062D:
		F_EtherCAT_VendorIDtoString := 'CG Drives & Automation AB';

	16#0000062E:
		F_EtherCAT_VendorIDtoString := 'ProCom GmbH';

	16#0000062F:
		F_EtherCAT_VendorIDtoString := 'ALSTOM Grid SAS - Systems';

	16#00000630:
		F_EtherCAT_VendorIDtoString := 'Robot Makers GmbH';

	16#00000631:
		F_EtherCAT_VendorIDtoString := 'Brooks Automation, Inc';

	16#00000632:
		F_EtherCAT_VendorIDtoString := 'Hitachi Metals Ltd., Piping Components Company';

	16#00000633:
		F_EtherCAT_VendorIDtoString := 'Interroll Automation GmbH';

	16#00000634:
		F_EtherCAT_VendorIDtoString := 'CKD Corporation';

	16#00000635:
		F_EtherCAT_VendorIDtoString := 'AMS Research GmbH';

	16#00000636:
		F_EtherCAT_VendorIDtoString := 'T.P.A. S.p.A';

	16#00000637:
		F_EtherCAT_VendorIDtoString := 'Guodian Nanjing Automation Co., Ltd.';

	16#00000638:
		F_EtherCAT_VendorIDtoString := 'Prosoft-Systems Ltd.';

	16#00000639:
		F_EtherCAT_VendorIDtoString := 'Polytype SA';

	16#0000063B:
		F_EtherCAT_VendorIDtoString := 'Delta Computer Systems, Inc.';

	16#0000063C:
		F_EtherCAT_VendorIDtoString := 'Friedrich Lütze GmbH';

	16#0000063D:
		F_EtherCAT_VendorIDtoString := 'Compressor Controls Corporation';

	16#0000063E:
		F_EtherCAT_VendorIDtoString := 'Diamond Light Source Limited';

	16#0000063F:
		F_EtherCAT_VendorIDtoString := 'Beckman Coulter, Inc.';

	16#00000641:
		F_EtherCAT_VendorIDtoString := 'Nor-Cal Products, Inc.';

	16#00000642:
		F_EtherCAT_VendorIDtoString := 'AUTOMATA GmbH & Co. KG';

	16#00000643:
		F_EtherCAT_VendorIDtoString := 'Fraunhofer Institut für Werkstoff- und Strahlentechnik IWS';

	16#00000644:
		F_EtherCAT_VendorIDtoString := 'INFICON AG';

	16#00000645:
		F_EtherCAT_VendorIDtoString := 'Hexagon Metrology GmbH';

	16#00000646:
		F_EtherCAT_VendorIDtoString := 'Shimadzu Corporation';

	16#00000647:
		F_EtherCAT_VendorIDtoString := 'Dasa Control Systems AB';

	16#00000648:
		F_EtherCAT_VendorIDtoString := 'SHOEI Electric Co.,Ltd.';

	16#00000649:
		F_EtherCAT_VendorIDtoString := 'Progressio, LLC';

	16#0000064A:
		F_EtherCAT_VendorIDtoString := 'MACCON GmbH';

	16#0000064B:
		F_EtherCAT_VendorIDtoString := 'Moog Ireland, Ltd.';

	16#0000064C:
		F_EtherCAT_VendorIDtoString := 'ESPERA-WERKE GMBH';

	16#0000064D:
		F_EtherCAT_VendorIDtoString := 'Automation W+R GmbH';

	16#0000064F:
		F_EtherCAT_VendorIDtoString := 'EOStech S.r.l.';

	16#00000650:
		F_EtherCAT_VendorIDtoString := 'Lycée Jean-Baptiste de Baudre';

	16#00000651:
		F_EtherCAT_VendorIDtoString := 'University of Banja Luka';

	16#00000652:
		F_EtherCAT_VendorIDtoString := 'Eding CNC';

	16#00000653:
		F_EtherCAT_VendorIDtoString := 'Zühlke Engineering AG';

	16#00000654:
		F_EtherCAT_VendorIDtoString := 'Addiva Consulting AB';

	16#00000655:
		F_EtherCAT_VendorIDtoString := 'Pteris Global Limited';

	16#00000656:
		F_EtherCAT_VendorIDtoString := 'Chaos Technology';

	16#00000657:
		F_EtherCAT_VendorIDtoString := 'Tokyo Institute of Technology, Hirose Fukushima Lab.';

	16#00000658:
		F_EtherCAT_VendorIDtoString := 'Seichter GmbH';

	16#00000659:
		F_EtherCAT_VendorIDtoString := 'Motion Control Systems, Inc.';

	16#0000065A:
		F_EtherCAT_VendorIDtoString := 'Moog B.V. in the Netherlands';

	16#0000065B:
		F_EtherCAT_VendorIDtoString := 'Kinlo Technology & System (Shenzhen) Co.,Ltd.';

	16#0000065C:
		F_EtherCAT_VendorIDtoString := 'CellSystems, LLC';

	16#0000065D:
		F_EtherCAT_VendorIDtoString := 'Shinano Kenshi Co., Ltd.';

	16#0000065E:
		F_EtherCAT_VendorIDtoString := 'MICRO-EPSILON MESSTECHNIK GmbH & Co. KG';

	16#0000065F:
		F_EtherCAT_VendorIDtoString := 'Viable Bytes, Inc.';

	16#00000660:
		F_EtherCAT_VendorIDtoString := 'Kontron AG';

	16#00000661:
		F_EtherCAT_VendorIDtoString := 'IKERLAN-IK4';

	16#00000662:
		F_EtherCAT_VendorIDtoString := 'hmk Daten-System-Technik GmbH';

	16#00000663:
		F_EtherCAT_VendorIDtoString := 'Wecon Automation Corp.';

	16#00000664:
		F_EtherCAT_VendorIDtoString := 'Istituto Italiano di Tecnologia (IIT)';

	16#00000665:
		F_EtherCAT_VendorIDtoString := 'Kashiyama Industries, Ltd.';

	16#00000666:
		F_EtherCAT_VendorIDtoString := 'TG Drives s.r.o.';

	16#00000667:
		F_EtherCAT_VendorIDtoString := 'Watlow Electric Manufacturing Company';

	16#00000668:
		F_EtherCAT_VendorIDtoString := 'synertronixx GmbH';

	16#00000669:
		F_EtherCAT_VendorIDtoString := 'batalpha Bobach GmbH';

	16#0000066A:
		F_EtherCAT_VendorIDtoString := 'Edwards Limited';

	16#0000066B:
		F_EtherCAT_VendorIDtoString := 'ENGEL AUSTRIA GmbH';

	16#0000066C:
		F_EtherCAT_VendorIDtoString := 'Fujikin Incorporated';

	16#0000066D:
		F_EtherCAT_VendorIDtoString := 'COMET Technologies USA, Inc.';

	16#0000066E:
		F_EtherCAT_VendorIDtoString := 'Schleuniger AG';

	16#0000066F:
		F_EtherCAT_VendorIDtoString := 'Panasonic Corporation, Appliances Company';

	16#00000670:
		F_EtherCAT_VendorIDtoString := 'TangShan Kaiyuan Welding Automation Technology Institute Co., Ltd.';

	16#00000671:
		F_EtherCAT_VendorIDtoString := 'Solectrix GmbH';

	16#00000672:
		F_EtherCAT_VendorIDtoString := 'St. Cloud State University, Electrical and Computer Engineering Department';

	16#00000673:
		F_EtherCAT_VendorIDtoString := 'JLG AUTOMATION BVBA';

	16#00000674:
		F_EtherCAT_VendorIDtoString := 'Burckhardt Compression AG';

	16#00000675:
		F_EtherCAT_VendorIDtoString := 'Rong Shun Xuan Corp.';

	16#00000676:
		F_EtherCAT_VendorIDtoString := 'STM Sensor Technologie München GmbH';

	16#00000677:
		F_EtherCAT_VendorIDtoString := 'Endress+Hauser Flowtec AG';

	16#00000678:
		F_EtherCAT_VendorIDtoString := 'Motor Power Company S.r.l.';

	16#0000067A:
		F_EtherCAT_VendorIDtoString := 'EBI Electric Inc.';

	16#0000067B:
		F_EtherCAT_VendorIDtoString := 'Hochschule Luzern - Technik & Architektur';

	16#0000067C:
		F_EtherCAT_VendorIDtoString := 'GE Global Research';

	16#0000067D:
		F_EtherCAT_VendorIDtoString := 'Katholieke Universiteit Leuven, Department of Mechanical Engineering';

	16#0000067E:
		F_EtherCAT_VendorIDtoString := 'Ectronic GmbH';

	16#0000067F:
		F_EtherCAT_VendorIDtoString := 'Bundesamt für Wehrtechnik und Beschaffung, Dienststelle WTD 81';

	16#00000680:
		F_EtherCAT_VendorIDtoString := 'DAIHEN Corporation';

	16#00000681:
		F_EtherCAT_VendorIDtoString := 'HCL Technologies Ltd.';

	16#00000682:
		F_EtherCAT_VendorIDtoString := '3T B.V.';

	16#00000683:
		F_EtherCAT_VendorIDtoString := 'Eindhoven University of Technology';

	16#00000685:
		F_EtherCAT_VendorIDtoString := 'Surrey Satellite Technology Limited';

	16#00000686:
		F_EtherCAT_VendorIDtoString := 'AMETEK Programmable Power, Inc.';

	16#00000687:
		F_EtherCAT_VendorIDtoString := 'engleder embedded';

	16#00000688:
		F_EtherCAT_VendorIDtoString := 'Pusan National University, Department of Intelligent Mechanical Engineering';

	16#00000689:
		F_EtherCAT_VendorIDtoString := 'ETH Zürich, D-HEST, Institute of Robotics and Intelligent Systems';

	16#0000068A:
		F_EtherCAT_VendorIDtoString := 'Berner & Mattner Systemtechnik GmbH';

	16#0000068B:
		F_EtherCAT_VendorIDtoString := 'HORIBA, Ltd.';

	16#0000068D:
		F_EtherCAT_VendorIDtoString := 'Penko Engineering B.V.';

	16#0000068E:
		F_EtherCAT_VendorIDtoString := 'Fujitsu Semiconductor Europe GmbH';

	16#00000690:
		F_EtherCAT_VendorIDtoString := 'Mirle Automation Corporation';

	16#00000691:
		F_EtherCAT_VendorIDtoString := 'FANUC CORPORATION';

	16#00000692:
		F_EtherCAT_VendorIDtoString := 'KSE GmbH';

	16#00000693:
		F_EtherCAT_VendorIDtoString := 'EUCHNER GmbH + Co. KG';

	16#00000694:
		F_EtherCAT_VendorIDtoString := 'benjamin GmbH';

	16#00000695:
		F_EtherCAT_VendorIDtoString := 'Hans Laser Technology Co.,Ltd.';

	16#00000696:
		F_EtherCAT_VendorIDtoString := 'Guangdong University of Technology, Faculty of Automation';

	16#00000699:
		F_EtherCAT_VendorIDtoString := 'Instituto Federal de Santa Catarina';

	16#0000069A:
		F_EtherCAT_VendorIDtoString := 'InstruTech Inc.';

	16#0000069B:
		F_EtherCAT_VendorIDtoString := 'KTL Corporation';

	16#0000069D:
		F_EtherCAT_VendorIDtoString := 'EWM HIGHTEC WELDING GmbH';

	16#0000069E:
		F_EtherCAT_VendorIDtoString := 'Jilin Yongda Group Company Ltd.';

	16#0000069F:
		F_EtherCAT_VendorIDtoString := 'Arrow Central Europe GmbH';

	16#00000700:
		F_EtherCAT_VendorIDtoString := 'Institut de RadioAstronomie Millimétrique';

	16#00000701:
		F_EtherCAT_VendorIDtoString := 'Technische Universität Graz, Fakultät für Maschinenbau und Wirtschaftswissenschaften';

	16#00000702:
		F_EtherCAT_VendorIDtoString := 'pro-beam AG & Co. KGaA';

	16#00000703:
		F_EtherCAT_VendorIDtoString := 'Servotechnica ZAO';

	16#00000704:
		F_EtherCAT_VendorIDtoString := 'Samsung Techwin Co. Ltd.';

	16#00000705:
		F_EtherCAT_VendorIDtoString := 'Softlink Technologies Co., Ltd.';

	16#00000706:
		F_EtherCAT_VendorIDtoString := 'Schaeffler Engineering';

	16#00000707:
		F_EtherCAT_VendorIDtoString := 'University of the Basque Country, Faculty of Engineering, Department of Electronics and Telecommunications';

	16#00000708:
		F_EtherCAT_VendorIDtoString := 'ARGES GmbH';

	16#00000709:
		F_EtherCAT_VendorIDtoString := 'Control Chief Corporation';

	16#0000070A:
		F_EtherCAT_VendorIDtoString := 'konplan systemhaus ag';

	16#0000070B:
		F_EtherCAT_VendorIDtoString := 'embeX GmbH';

	16#0000070C:
		F_EtherCAT_VendorIDtoString := 'COSMOTECHS Co., Ltd';

	16#0000070D:
		F_EtherCAT_VendorIDtoString := 'Dynamic Systems Inc.';

	16#0000070E:
		F_EtherCAT_VendorIDtoString := 'SEMIKRON Elektronik GmbH & Co. KG';

	16#0000070F:
		F_EtherCAT_VendorIDtoString := 'Wuxi Ivoyage Control Technology CO.,LTD';

	16#00000710:
		F_EtherCAT_VendorIDtoString := 'CAF Signalling S.L.';

	16#00000711:
		F_EtherCAT_VendorIDtoString := 'SMART Electronic Development GmbH';

	16#00000712:
		F_EtherCAT_VendorIDtoString := 'Yokogawa Electric Corporation';

	16#00000713:
		F_EtherCAT_VendorIDtoString := 'Norwegian University of Science and Technoloogy, Faculty of Information Technology, Mathematics and Electrical Engineering';

	16#00000715:
		F_EtherCAT_VendorIDtoString := 'TRUMPF Werkzeugmaschinen GmbH + Co. KG';

	16#00000716:
		F_EtherCAT_VendorIDtoString := 'High Performance Motion System Development Co., Ltd.';

	16#00000717:
		F_EtherCAT_VendorIDtoString := 'Kozaka Electronic Design Inc.';

	16#00000718:
		F_EtherCAT_VendorIDtoString := 'Aeronautical Systems Engineering Inc.';

	16#00000719:
		F_EtherCAT_VendorIDtoString := 'Agile Planet, Inc.';

	16#0000071A:
		F_EtherCAT_VendorIDtoString := 'Hon Hai Precision Industry Co., Ltd.';

	16#0000071B:
		F_EtherCAT_VendorIDtoString := 'Systeme + Steuerungen GmbH';

	16#0000071C:
		F_EtherCAT_VendorIDtoString := 'Huron Net Works, Inc.';

	16#0000071D:
		F_EtherCAT_VendorIDtoString := 'University of Applied Sciences of Southern Switzerland, Department of Innovative Technologies (DTI)';

	16#0000071E:
		F_EtherCAT_VendorIDtoString := 'MAKO Surgical Corp.';

	16#0000071F:
		F_EtherCAT_VendorIDtoString := 'Rainer Thomas Messtechnik GmbH';

	16#00000720:
		F_EtherCAT_VendorIDtoString := 'ELTEK spol. s r.o.';

	16#00000721:
		F_EtherCAT_VendorIDtoString := 'Vecow Co., Ltd.';

	16#00000722:
		F_EtherCAT_VendorIDtoString := 'M&P Motion Control and Power Electronics GmbH';

	16#00000723:
		F_EtherCAT_VendorIDtoString := 'Oerlikon Leybold Vacuum GmbH';

	16#00000725:
		F_EtherCAT_VendorIDtoString := 'Panasonic Electric Works Corporation of America';

	16#00000726:
		F_EtherCAT_VendorIDtoString := 'Eilersen Electric Digital Systems A/S';

	16#00000727:
		F_EtherCAT_VendorIDtoString := 'Inter Factory Partners Co., LTD.';

	16#00000728:
		F_EtherCAT_VendorIDtoString := 'Power Instrument Co., Ltd.';

	16#00000729:
		F_EtherCAT_VendorIDtoString := 'Cosworth Group Holdings Ltd';

	16#0000072A:
		F_EtherCAT_VendorIDtoString := 'South China University of Technology, School of Mechanical & Automotive Engineering';

	16#0000072B:
		F_EtherCAT_VendorIDtoString := 'WARWICK INSTRUMENTS LTD.';

	16#0000072C:
		F_EtherCAT_VendorIDtoString := 'Shenzhen INVT Co., Ltd.';

	16#0000072D:
		F_EtherCAT_VendorIDtoString := 'WIEDEG Elektronik GmbH';

	16#0000072E:
		F_EtherCAT_VendorIDtoString := 'NKE corporation';

	16#0000072F:
		F_EtherCAT_VendorIDtoString := 'Universidad Politécnica de Madrid';

	16#00000730:
		F_EtherCAT_VendorIDtoString := 'Bot & Dolly';

	16#00000731:
		F_EtherCAT_VendorIDtoString := 'RECIF Technologies';

	16#00000732:
		F_EtherCAT_VendorIDtoString := 'ATI Industrial Automation';

	16#00000734:
		F_EtherCAT_VendorIDtoString := 'Multivac Sepp Haggenmüller GmbH & Co. KG';

	16#00000735:
		F_EtherCAT_VendorIDtoString := 'ROLAND ELECTRONIC GmbH';

	16#00000736:
		F_EtherCAT_VendorIDtoString := 'CONTEC Co., Ltd.';

	16#00000737:
		F_EtherCAT_VendorIDtoString := 'Alizem Inc.';

	16#00000739:
		F_EtherCAT_VendorIDtoString := 'Yaskawa America Inc.';

	16#0000073B:
		F_EtherCAT_VendorIDtoString := 'Faraday Technology Corporation';

	16#0000073C:
		F_EtherCAT_VendorIDtoString := 'SIPRO S.r.l.';

	16#0000073D:
		F_EtherCAT_VendorIDtoString := 'University of Twente, Faculty of Engineering Technology (CTW)';

	16#0000073E:
		F_EtherCAT_VendorIDtoString := 'Aalborg University';

	16#0000073F:
		F_EtherCAT_VendorIDtoString := 'S-SYS bvba';

	16#00000740:
		F_EtherCAT_VendorIDtoString := 'Ningbo Mingpu Automation Technology Co.';

	16#00000741:
		F_EtherCAT_VendorIDtoString := 'elrest Automationssysteme GmbH';

	16#00000742:
		F_EtherCAT_VendorIDtoString := 'Kyosan Electric Manufacturing Co., Ltd.';

	16#00000743:
		F_EtherCAT_VendorIDtoString := 'Egret Engineering Pty Ltd';

	16#00000744:
		F_EtherCAT_VendorIDtoString := 'KFM Regelungstechnik GmbH';

	16#00000745:
		F_EtherCAT_VendorIDtoString := 'ISHIDA CO., LTD.';

	16#00000746:
		F_EtherCAT_VendorIDtoString := 'Beijing University of Technology';

	16#00000747:
		F_EtherCAT_VendorIDtoString := 'Hannifin Corporation, Electromechanical Automation Division, North America';

	16#00000748:
		F_EtherCAT_VendorIDtoString := 'Tsino-dynatron Electrical Technology Beijing Co., Ltd.';

	16#00000749:
		F_EtherCAT_VendorIDtoString := 'PENTA TRADING Spol. S.r.o.';

	16#0000074A:
		F_EtherCAT_VendorIDtoString := 'University of Electronic Science and Technology of China, School of Optoelectronic Information';

	16#0000074B:
		F_EtherCAT_VendorIDtoString := 'Altus Sistemas de Informática S/A';

	16#0000074C:
		F_EtherCAT_VendorIDtoString := 'Sanming University, Sanming Mechanical CAD Engineering Research Center';

	16#0000074E:
		F_EtherCAT_VendorIDtoString := 'Hommel-Etamic GmbH';

	16#0000074F:
		F_EtherCAT_VendorIDtoString := 'Beijing KND CNC Technique Co., Ltd.';

	16#00000750:
		F_EtherCAT_VendorIDtoString := 'JW Shannon Engineers';

	16#00000751:
		F_EtherCAT_VendorIDtoString := 'A2V Mécatronique SAS';

	16#00000752:
		F_EtherCAT_VendorIDtoString := 'NEXCOM International Co., Ltd.';

	16#00000753:
		F_EtherCAT_VendorIDtoString := 'Jiangyin Huafeng Printing Machinery Co., Ltd.';

	16#00000754:
		F_EtherCAT_VendorIDtoString := 'Lectra';

	16#00000755:
		F_EtherCAT_VendorIDtoString := 'Beijer Electronics Products AB';

	16#00000756:
		F_EtherCAT_VendorIDtoString := 'C J Hartman Elektronik AB';

	16#00000757:
		F_EtherCAT_VendorIDtoString := 'Hurco Automation Ltd.';

	16#00000759:
		F_EtherCAT_VendorIDtoString := 'Autonics Corporation';

	16#0000075A:
		F_EtherCAT_VendorIDtoString := 'Brom Mechatronica B.V.';

	16#0000075B:
		F_EtherCAT_VendorIDtoString := 'Vrije Universiteit Brussel, Faculty of Engineering';

	16#0000075C:
		F_EtherCAT_VendorIDtoString := 'Alluris GmbH & Co. KG';

	16#0000075D:
		F_EtherCAT_VendorIDtoString := 'Hochschule Offenburg, Fakultät Elektrotechnik und Informationstechnik';

	16#0000075F:
		F_EtherCAT_VendorIDtoString := 'Heidolph Elektro GmbH & Co. KG';

	16#00000760:
		F_EtherCAT_VendorIDtoString := 'GE Transportation';

	16#00000761:
		F_EtherCAT_VendorIDtoString := 'MÄX GmbH';

	16#00000762:
		F_EtherCAT_VendorIDtoString := 'Durst Phototechnik Digital Technology GmbH';

	16#00000763:
		F_EtherCAT_VendorIDtoString := 'Omsk State Technical University, Department of „Electricity industry“';

	16#00000764:
		F_EtherCAT_VendorIDtoString := 'Embedded-Bonjour GmbH';

	16#00000765:
		F_EtherCAT_VendorIDtoString := 'Mettler-Toledo Garvens GmbH';

	16#00000766:
		F_EtherCAT_VendorIDtoString := 'Renesas Electronics Corp.';

	16#00000767:
		F_EtherCAT_VendorIDtoString := 'LJU Automatisierungstechnik GmbH';

	16#00000768:
		F_EtherCAT_VendorIDtoString := 'EURA DRIVES ELECTRIC CO. LTD';

	16#00000769:
		F_EtherCAT_VendorIDtoString := 'EUTRON S.p.A.';

	16#0000076A:
		F_EtherCAT_VendorIDtoString := 'FLANDERS Inc.';

	16#0000076B:
		F_EtherCAT_VendorIDtoString := 'Digital Dynamics, Inc.';

	16#0000076C:
		F_EtherCAT_VendorIDtoString := 'GE Medical Systems Europe';

	16#0000076D:
		F_EtherCAT_VendorIDtoString := 'Physik Instumente GmbH & Co. KG';

	16#0000076E:
		F_EtherCAT_VendorIDtoString := 'Hypertherm Inc.';

	16#0000076F:
		F_EtherCAT_VendorIDtoString := 'HRID d.o.o.';

	16#00000770:
		F_EtherCAT_VendorIDtoString := 'Aotai Electric Co., LTD';

	16#00000771:
		F_EtherCAT_VendorIDtoString := 'Control Concepts Inc.';

	16#00000772:
		F_EtherCAT_VendorIDtoString := 'JoveTech Co., Ltd.';

	16#00000773:
		F_EtherCAT_VendorIDtoString := 'POHANG UNIVERSITY OF SCIENCE AND TECHNOLOGY, Department of Electrical Engineering';

	16#00000774:
		F_EtherCAT_VendorIDtoString := 'CycloMedia Technology B.V.';

	16#00000775:
		F_EtherCAT_VendorIDtoString := 'SUN-TECTRO LTD.';

	16#00000776:
		F_EtherCAT_VendorIDtoString := 'Shanghai Jiao Tong University, School of Electronic Information and Electrical Engineering';

	16#00000777:
		F_EtherCAT_VendorIDtoString := 'koenig-pa GmbH';

	16#00000778:
		F_EtherCAT_VendorIDtoString := 'CSM Instruments SA';

	16#00000779:
		F_EtherCAT_VendorIDtoString := 'V TEX Corporation';

	16#0000077A:
		F_EtherCAT_VendorIDtoString := 'Edge Technologies';

	16#0000077B:
		F_EtherCAT_VendorIDtoString := 'EBARA CORPORATION';

	16#0000077C:
		F_EtherCAT_VendorIDtoString := 'University at Buffalo';

	16#0000077D:
		F_EtherCAT_VendorIDtoString := 'Aurotek Corporation';

	16#0000077E:
		F_EtherCAT_VendorIDtoString := 'Blubit d.o.o.';

	16#0000077F:
		F_EtherCAT_VendorIDtoString := 'Toplens Hangzhou, Inc.';

	16#00000782:
		F_EtherCAT_VendorIDtoString := 'Graph-Tech AG';

	16#00000783:
		F_EtherCAT_VendorIDtoString := 'Lanthan GmbH & Co. KG';

	16#00000784:
		F_EtherCAT_VendorIDtoString := 'Nucleus GmbH';

	16#00000785:
		F_EtherCAT_VendorIDtoString := 'STRATEC CONTROL-SYSTEMS GmbH';

	16#00000786:
		F_EtherCAT_VendorIDtoString := 'Universität Wien, Fakultät für Physik, Isotopenforschung';

	16#00000787:
		F_EtherCAT_VendorIDtoString := 'inno-spec GmbH';

	16#00000788:
		F_EtherCAT_VendorIDtoString := 'ThyssenKrupp Presta AG';

	16#0000078A:
		F_EtherCAT_VendorIDtoString := 'DENSO WAVE INCORPORATED';

	16#0000078B:
		F_EtherCAT_VendorIDtoString := 'EuroSoft S.r.l.';

	16#0000078C:
		F_EtherCAT_VendorIDtoString := 'University of British Columbia, Faculty of Applied Science, Department of Mechanical Engineering';

	16#0000078D:
		F_EtherCAT_VendorIDtoString := 'REnergy Electric Tianjin Ltd.';

	16#0000078E:
		F_EtherCAT_VendorIDtoString := 'NewYoungSystem Co., Ltd.';

	16#0000078F:
		F_EtherCAT_VendorIDtoString := 'Selema S.r.l.';

	16#00000790:
		F_EtherCAT_VendorIDtoString := 'University of Reading, School of Systems Engineering';

	16#00000791:
		F_EtherCAT_VendorIDtoString := 'KOGANEI CORPORATION';

	16#00000792:
		F_EtherCAT_VendorIDtoString := 'MAZeT GmbH';

	16#00000793:
		F_EtherCAT_VendorIDtoString := 'The University of Nottingham, Faculty of Engineering, Electrical Systems and Optics Research Division';

	16#00000794:
		F_EtherCAT_VendorIDtoString := 'Quanta Storage Inc.';

	16#00000795:
		F_EtherCAT_VendorIDtoString := 'Azbil Taishin Co., Ltd.';

	16#00000796:
		F_EtherCAT_VendorIDtoString := 'Relitech B.V.';

	16#00000797:
		F_EtherCAT_VendorIDtoString := 'DHPC Technologies, Inc.';

	16#00000798:
		F_EtherCAT_VendorIDtoString := 'Jordan Valley Semiconductors Ltd.';

	16#00000799:
		F_EtherCAT_VendorIDtoString := 'MicroCreate System Co., Ltd.';

	16#0000079A:
		F_EtherCAT_VendorIDtoString := 'AB&T S.r.l.';

	16#0000079C:
		F_EtherCAT_VendorIDtoString := 'T3LAB - Technology Transfer Team';

	16#0000079D:
		F_EtherCAT_VendorIDtoString := 'Coptonix GmbH';

	16#0000079E:
		F_EtherCAT_VendorIDtoString := 'KARL MAYER Textilmaschinenfabrik GmbH';

	16#0000079F:
		F_EtherCAT_VendorIDtoString := 'inoson GmbH';

	16#00000801:
		F_EtherCAT_VendorIDtoString := 'OTSL Inc.';

	16#00000802:
		F_EtherCAT_VendorIDtoString := 'Aromasoft Corp.';

	16#0000089E:
		F_EtherCAT_VendorIDtoString := 'D2T SA';

	16#000008E7:
		F_EtherCAT_VendorIDtoString := 'Sumitomo Heavy Industries, Ltd.';

	16#00000900:
		F_EtherCAT_VendorIDtoString := 'Shanghai Capital Numerical Control Co., Ltd.';

	16#00000999:
		F_EtherCAT_VendorIDtoString := 'HAITIAN Plastics Machinery Group Co., Ltd';

	16#00000A1E:
		F_EtherCAT_VendorIDtoString := 'Mitsubishi Electric Corporation';

	16#00000ABB:
		F_EtherCAT_VendorIDtoString := 'ABB AS Corporate Research';

	16#00000AFA:
		F_EtherCAT_VendorIDtoString := 'Afag Automation AG';

	16#00000D05:
		F_EtherCAT_VendorIDtoString := 'John Deere Werke Mannheim';

	16#00000D0F:
		F_EtherCAT_VendorIDtoString := 'DEIF A/S';

	16#000010FA:
		F_EtherCAT_VendorIDtoString := 'Beijing BBF Servo Technology Co.,Ltd.';

	16#00001110:
		F_EtherCAT_VendorIDtoString := 'A-KYUNG Motion Inc.';

	16#00001111:
		F_EtherCAT_VendorIDtoString := 'MLS Lanny GmbH';

	16#00001122:
		F_EtherCAT_VendorIDtoString := 'CanTops';

	16#000012AD:
		F_EtherCAT_VendorIDtoString := 'IDS GmbH';

	16#00001337:
		F_EtherCAT_VendorIDtoString := 'rt-labs AB';

	16#000013FE:
		F_EtherCAT_VendorIDtoString := 'Advantech Co., Ltd.';

	16#0000144A:
		F_EtherCAT_VendorIDtoString := 'ADLINK TECHNOLOGY INC.';

	16#0000147A:
		F_EtherCAT_VendorIDtoString := 'eubus GmbH';

	16#00001502:
		F_EtherCAT_VendorIDtoString := 'Unico Inc.';

	16#00001600:
		F_EtherCAT_VendorIDtoString := 'Helmholtz-Zentrum Dresden-Rossendorf e.V.';

	16#00001616:
		F_EtherCAT_VendorIDtoString := 'DLR Deutsches Zentrum für Luft- und Raumfahrt e.V.';

	16#00001701:
		F_EtherCAT_VendorIDtoString := 'PLR Prüftechnik Linke & Rühe GmbH';

	16#0000179A:
		F_EtherCAT_VendorIDtoString := 'Haute Ecole dIngénierie et de Gestion du Canton de Vaud du Canton de Vaud';

	16#00001800:
		F_EtherCAT_VendorIDtoString := 'TAMAGAWA SEIKI CO.,LTD.';

	16#00001899:
		F_EtherCAT_VendorIDtoString := 'Hagenuk Marinekommunikation GmbH';

	16#00001919:
		F_EtherCAT_VendorIDtoString := 'SACMI IMOLA S.C.';

	16#00001984:
		F_EtherCAT_VendorIDtoString := 'LAUMAS Elettronica s.r.l.';

	16#00001987:
		F_EtherCAT_VendorIDtoString := 'DINA Elektronik GmbH';

	16#00001A05:
		F_EtherCAT_VendorIDtoString := 'SYN-TEK Technologies Inc.';

	16#00001A21:
		F_EtherCAT_VendorIDtoString := 'BySTORM & CO. srl';

	16#00001A85:
		F_EtherCAT_VendorIDtoString := 'Michel Van de Wiele NV';

	16#00001A90:
		F_EtherCAT_VendorIDtoString := 'IPETRONIK GmbH & Co. KG';

	16#00001B2C:
		F_EtherCAT_VendorIDtoString := 'Opal-RT Technologies, Inc.';

	16#00001B66:
		F_EtherCAT_VendorIDtoString := 'Sennheiser electronic GmbH & Co. KG';

	16#000022D2:
		F_EtherCAT_VendorIDtoString := 'Synapticon GmbH';

	16#00002304:
		F_EtherCAT_VendorIDtoString := 'DANIELI AUTOMATION SPA';

	16#000027AB:
		F_EtherCAT_VendorIDtoString := 'Rollmann Elektronik';

	16#00002838:
		F_EtherCAT_VendorIDtoString := 'burster präzisionsmesstechnik gmbh & co kg';

	16#000033C3:
		F_EtherCAT_VendorIDtoString := 'MatrixGroup (CMS) Pty Ltd';

	16#00004154:
		F_EtherCAT_VendorIDtoString := 'acontis technologies GmbH';

	16#00004321:
		F_EtherCAT_VendorIDtoString := 'Leadshine Technology Co., Ltd.';

